C01817=1154.815,15.014,-48.250,179.930,6.144,149.128
C01818=1154.820,14.765,-48.236,179.927,6.143,149.129
C01819=1154.826,14.515,-48.222,179.924,6.142,149.129
C01820=1154.831,14.265,-48.208,179.922,6.141,149.130
C01821=1154.836,14.016,-48.194,179.919,6.140,149.130
C01822=1154.841,13.767,-48.180,179.917,6.140,149.131
C01823=1154.846,13.517,-48.166,179.915,6.139,149.131
C01824=1154.850,13.267,-48.152,179.911,6.138,149.132
C01825=1154.856,13.018,-48.139,179.909,6.137,149.133
C01826=1154.861,12.768,-48.125,179.906,6.137,149.133
C01827=1154.866,12.518,-48.110,179.904,6.136,149.134
C01828=1154.872,12.269,-48.096,179.902,6.135,149.134
C01829=1154.877,12.019,-48.083,179.899,6.134,149.135
C01830=1154.881,11.770,-48.069,179.896,6.133,149.136
C01831=1154.887,11.521,-48.055,179.894,6.132,149.136
C01832=1154.892,11.271,-48.041,179.891,6.132,149.137
C01833=1154.897,11.021,-48.027,179.889,6.131,149.137
C01834=1154.903,10.772,-48.013,179.887,6.131,149.138
C01835=1154.907,10.522,-48.000,179.884,6.129,149.138
C01836=1154.913,10.273,-47.987,179.881,6.129,149.139
C01837=1154.918,10.023,-47.972,179.879,6.128,149.139
C01838=1154.923,9.773,-47.958,179.876,6.127,149.140
C01839=1154.928,9.524,-47.945,179.874,6.127,149.141
C01840=1154.933,9.274,-47.931,179.871,6.125,149.141
C01841=1154.938,9.024,-47.917,179.869,6.125,149.142
C01842=1154.943,8.775,-47.904,179.866,6.124,149.142
C01843=1154.948,8.525,-47.890,179.864,6.123,149.143
C01844=1154.953,8.276,-47.876,179.861,6.123,149.144
C01845=1154.959,8.026,-47.862,179.859,6.122,149.144
C01846=1154.963,7.777,-47.849,179.856,6.121,149.145
C01847=1154.969,7.527,-47.836,179.854,6.120,149.145
C01848=1154.974,7.277,-47.821,179.851,6.119,149.146
C01849=1154.979,7.028,-47.807,179.849,6.119,149.146
C01850=1154.984,6.778,-47.794,179.846,6.118,149.147
C01851=1154.989,6.529,-47.781,179.844,6.117,149.147
C01852=1154.994,6.279,-47.767,179.841,6.116,149.148
C01853=1154.999,6.030,-47.754,179.839,6.115,149.149
C01854=1155.005,5.780,-47.740,179.836,6.115,149.149
C01855=1155.009,5.530,-47.726,179.834,6.114,149.150
C01856=1155.015,5.281,-47.713,179.831,6.114,149.150
C01857=1155.020,5.031,-47.699,179.829,6.113,149.151
C01858=1155.025,4.782,-47.686,179.826,6.111,149.152
C01859=1155.030,4.532,-47.672,179.824,6.111,149.152
C01860=1155.036,4.283,-47.659,179.821,6.110,149.153
C01861=1155.040,4.033,-47.645,179.819,6.109,149.153
C01862=1155.046,3.784,-47.632,179.816,6.109,149.154
C01863=1155.050,3.534,-47.618,179.814,6.108,149.154
C01864=1155.056,3.284,-47.605,179.811,6.108,149.155
C01865=1155.061,3.035,-47.591,179.808,6.106,149.155
C01866=1155.066,2.785,-47.578,179.806,6.106,149.156
C01867=1155.071,2.536,-47.564,179.804,6.105,149.157
C01868=1155.076,2.286,-47.551,179.801,6.104,149.157
C01869=1155.081,2.017,-47.536,179.799,6.104,149.158
C01870=1155.087,1.747,-47.522,179.796,6.102,149.158
C01871=1155.092,1.478,-47.507,179.793,6.102,149.159
C01872=1155.098,1.209,-47.494,179.790,6.101,149.160
C01873=1155.103,0.959,-47.479,179.788,6.101,149.160
C01874=1155.108,0.710,-47.467,179.785,6.100,149.161
C01875=1155.113,0.459,-47.453,179.783,6.099,149.161
C01876=1155.119,0.210,-47.439,179.780,6.098,149.162
C01877=1155.123,-0.040,-47.426,179.778,6.097,149.163
C01878=1155.129,-0.289,-47.413,179.775,6.097,149.163
C01879=1155.134,-0.539,-47.400,179.773,6.096,149.164
C01880=1155.139,-0.789,-47.386,179.770,6.096,149.164
C01881=1155.145,-1.038,-47.374,179.768,6.095,149.165
C01882=1155.149,-1.288,-47.360,179.766,6.094,149.166
C01883=1155.155,-1.537,-47.347,179.763,6.093,149.166
C01884=1155.160,-1.787,-47.333,179.760,6.092,149.167
C01885=1155.165,-2.036,-47.320,179.758,6.091,149.167
C01886=1155.169,-2.286,-47.307,179.755,6.091,149.168
C01887=1155.175,-2.536,-47.294,179.753,6.090,149.168
C01888=1155.180,-2.785,-47.281,179.750,6.090,149.169
C01889=1155.185,-3.035,-47.267,179.748,6.089,149.170
C01890=1155.190,-3.284,-47.254,179.746,6.088,149.170
C01891=1155.196,-3.534,-47.241,179.743,6.088,149.171
C01892=1155.201,-3.784,-47.228,179.741,6.087,149.171
C01893=1155.206,-4.033,-47.215,179.738,6.086,149.172
C01894=1155.211,-4.283,-47.201,179.735,6.085,149.173
C01895=1155.216,-4.532,-47.189,179.733,6.084,149.173
C01896=1155.221,-4.782,-47.175,179.731,6.084,149.174
C01897=1155.226,-5.032,-47.163,179.728,6.083,149.174
C01898=1155.232,-5.281,-47.149,179.726,6.083,149.175
C01899=1155.237,-5.531,-47.136,179.724,6.082,149.175
C01900=1155.241,-5.780,-47.123,179.721,6.081,149.176
C01901=1155.247,-6.029,-47.110,179.719,6.081,149.176
C01902=1155.252,-6.280,-47.097,179.716,6.080,149.177
C01903=1155.257,-6.529,-47.084,179.714,6.079,149.178
C01904=1155.263,-6.778,-47.071,179.711,6.079,149.178
C01905=1155.267,-7.028,-47.058,179.708,6.077,149.179
C01906=1155.273,-7.278,-47.045,179.706,6.077,149.179
C01907=1155.278,-7.527,-47.032,179.704,6.076,149.180
C01908=1155.283,-7.777,-47.019,179.701,6.076,149.181
C01909=1155.289,-8.027,-47.006,179.699,6.075,149.181
C01910=1155.294,-8.276,-46.993,179.696,6.074,149.182
C01911=1155.298,-8.526,-46.980,179.694,6.074,149.182
C01912=1155.303,-8.775,-46.967,179.691,6.073,149.183
C01913=1155.309,-9.025,-46.954,179.689,6.072,149.183
C01914=1155.314,-9.275,-46.941,179.686,6.072,149.184
C01915=1155.319,-9.524,-46.929,179.684,6.071,149.185
C01916=1155.325,-9.774,-46.915,179.682,6.071,149.185
C01917=1155.329,-10.024,-46.902,179.679,6.070,149.186
C01918=1155.334,-10.273,-46.890,179.677,6.069,149.186
C01919=1155.339,-10.522,-46.877,179.674,6.068,149.187
C01920=1155.345,-10.773,-46.864,179.671,6.067,149.188
C01921=1155.350,-11.022,-46.851,179.669,6.066,149.188
C01922=1155.355,-11.271,-46.838,179.666,6.066,149.189
C01923=1155.360,-11.521,-46.826,179.664,6.065,149.189
C01924=1155.365,-11.771,-46.812,179.662,6.065,149.190
C01925=1155.371,-12.021,-46.800,179.659,6.064,149.190
C01926=1155.376,-12.270,-46.788,179.657,6.064,149.191
C01927=1155.380,-12.520,-46.775,179.655,6.063,149.192
C01928=1155.386,-12.770,-46.762,179.652,6.062,149.192
C01929=1155.391,-13.019,-46.749,179.650,6.061,149.193
C01930=1155.396,-13.268,-46.736,179.647,6.061,149.193
C01931=1155.401,-13.519,-46.723,179.645,6.060,149.194
C01932=1155.406,-13.768,-46.711,179.642,6.060,149.195
C01933=1155.412,-14.017,-46.698,179.640,6.059,149.195
C01934=1155.417,-14.267,-46.685,179.637,6.059,149.196
C01935=1155.422,-14.517,-46.673,179.635,6.058,149.196
C01936=1155.427,-14.767,-46.660,179.633,6.057,149.197
C01937=1155.432,-15.016,-46.648,179.630,6.057,149.197
C01938=1155.437,-15.265,-46.635,179.628,6.056,149.198
C01939=1155.443,-15.515,-46.622,179.626,6.055,149.198
C01940=1155.448,-15.765,-46.609,179.623,6.055,149.199
C01941=1155.453,-16.015,-46.597,179.621,6.054,149.200
C01942=1155.458,-16.264,-46.584,179.618,6.054,149.200
C01943=1155.463,-16.514,-46.572,179.615,6.052,149.201
C01944=1155.468,-16.763,-46.559,179.613,6.052,149.201
C01945=1155.473,-17.014,-46.547,179.611,6.051,149.202
C01946=1155.478,-17.263,-46.534,179.608,6.050,149.203
C01947=1155.484,-17.512,-46.521,179.606,6.050,149.203
C01948=1155.489,-17.762,-46.509,179.603,6.049,149.204
C01949=1155.495,-18.012,-46.497,179.601,6.048,149.204
C01950=1155.500,-18.261,-46.484,179.598,6.048,149.205
C01951=1155.504,-18.511,-46.471,179.596,6.047,149.205
C01952=1155.510,-18.760,-46.458,179.593,6.047,149.206
C01953=1155.515,-19.010,-46.447,179.591,6.046,149.207
C01954=1155.520,-19.260,-46.434,179.588,6.045,149.207
C01955=1155.525,-19.509,-46.421,179.586,6.045,149.208
C01956=1155.531,-19.759,-46.409,179.584,6.044,149.208
C01957=1155.535,-20.009,-46.397,179.581,6.043,149.209
C01958=1155.540,-20.258,-46.384,179.579,6.043,149.210
C01959=1155.546,-20.508,-46.372,179.577,6.042,149.210
C01960=1155.551,-20.757,-46.359,179.574,6.042,149.211
C01961=1155.556,-21.007,-46.347,179.572,6.041,149.211
C01962=1155.562,-21.257,-46.334,179.569,6.040,149.212
C01963=1155.567,-21.506,-46.322,179.566,6.040,149.213
C01964=1155.572,-21.756,-46.309,179.564,6.039,149.213
C01965=1155.577,-22.006,-46.297,179.562,6.039,149.214
C01966=1155.582,-22.256,-46.284,179.559,6.038,149.214
C01967=1155.588,-22.506,-46.272,179.557,6.038,149.215
C01968=1155.593,-22.755,-46.260,179.555,6.037,149.215
C01969=1155.598,-23.004,-46.247,179.552,6.036,149.216
C01970=1155.603,-23.254,-46.235,179.550,6.036,149.217
C01971=1155.609,-23.503,-46.223,179.547,6.035,149.217
C01972=1155.613,-23.753,-46.211,179.545,6.034,149.218
C01973=1155.619,-24.023,-46.197,179.542,6.034,149.219
C01974=1155.625,-24.293,-46.185,179.540,6.033,149.219
C01975=1155.630,-24.563,-46.172,179.537,6.033,149.220
C01976=1155.636,-24.833,-46.157,179.535,6.032,149.220
C01977=1155.641,-25.083,-46.146,179.533,6.031,149.221
C01978=1155.646,-25.332,-46.133,179.530,6.031,149.222
C01979=1155.651,-25.582,-46.122,179.528,6.030,149.222
C01980=1155.656,-25.831,-46.109,179.525,6.030,149.223
C01981=1155.662,-26.081,-46.097,179.523,6.029,149.223
C01982=1155.667,-26.331,-46.084,179.520,6.029,149.224
C01983=1155.672,-26.581,-46.073,179.518,6.028,149.224
C01984=1155.677,-26.830,-46.060,179.515,6.027,149.225
C01985=1155.683,-27.080,-46.048,179.513,6.027,149.226
C01986=1155.688,-27.330,-46.036,179.511,6.026,149.226
C01987=1155.693,-27.579,-46.024,179.508,6.025,149.227
C01988=1155.698,-27.829,-46.012,179.506,6.025,149.227
C01989=1155.703,-28.078,-46.000,179.504,6.024,149.228
C01990=1155.709,-28.328,-45.988,179.501,6.024,149.229
C01991=1155.714,-28.577,-45.975,179.499,6.023,149.229
C01992=1155.719,-28.827,-45.963,179.496,6.022,149.230
C01993=1155.725,-29.077,-45.951,179.494,6.022,149.230
C01994=1155.729,-29.326,-45.939,179.492,6.022,149.231
C01995=1155.734,-29.576,-45.928,179.490,6.021,149.231
C01996=1155.740,-29.826,-45.916,179.487,6.021,149.232
C01997=1155.745,-30.075,-45.903,179.485,6.020,149.233
C01998=1155.750,-30.325,-45.891,179.482,6.020,149.233
C01999=1155.755,-30.575,-45.880,179.480,6.019,149.234
C02000=1155.760,-30.824,-45.867,179.477,6.018,149.234
C02001=1155.766,-31.074,-45.855,179.475,6.018,149.235
C02002=1155.771,-31.324,-45.844,179.472,6.017,149.236
C02003=1155.776,-31.573,-45.831,179.470,6.016,149.236
C02004=1155.781,-31.823,-45.820,179.468,6.016,149.237
C02005=1155.786,-32.073,-45.808,179.465,6.015,149.237
C02006=1155.791,-32.322,-45.795,179.463,6.015,149.238
C02007=1155.797,-32.572,-45.783,179.461,6.014,149.238
C02008=1155.802,-32.822,-45.772,179.458,6.013,149.239
C02009=1155.807,-33.072,-45.760,179.456,6.013,149.240
C02010=1155.812,-33.321,-45.747,179.453,6.012,149.240
C02011=1155.818,-33.571,-45.736,179.451,6.012,149.241
C02012=1155.822,-33.821,-45.724,179.449,6.012,149.241
C02013=1155.828,-34.071,-45.712,179.447,6.011,149.242
C02014=1155.833,-34.320,-45.700,179.444,6.011,149.243
C02015=1155.838,-34.570,-45.688,179.442,6.010,149.243
C02016=1155.843,-34.820,-45.677,179.439,6.009,149.244
C02017=1155.849,-35.069,-45.665,179.437,6.009,149.244
C02018=1155.854,-35.319,-45.653,179.434,6.008,149.245
C02019=1155.859,-35.568,-45.641,179.432,6.007,149.245
C02020=1155.864,-35.818,-45.629,179.429,6.007,149.246
C02021=1155.870,-36.068,-45.617,179.427,6.006,149.247
C02022=1155.875,-36.317,-45.606,179.425,6.006,149.247
C02023=1155.880,-36.567,-45.594,179.423,6.006,149.248
C02024=1155.885,-36.817,-45.582,179.420,6.005,149.248
C02025=1155.891,-37.067,-45.571,179.418,6.005,149.249
C02026=1155.896,-37.315,-45.559,179.416,6.004,149.249
C02027=1155.901,-37.565,-45.547,179.413,6.003,149.250
C02028=1155.906,-37.815,-45.535,179.411,6.003,149.251
C02029=1155.911,-38.065,-45.524,179.408,6.002,149.251
C02030=1155.917,-38.315,-45.512,179.406,6.001,149.252
C02031=1155.921,-38.564,-45.501,179.404,6.001,149.252
C02032=1155.927,-38.814,-45.489,179.401,6.000,149.253
C02033=1155.932,-39.064,-45.477,179.399,6.000,149.254
C02034=1155.937,-39.313,-45.466,179.397,6.000,149.254
C02035=1155.943,-39.563,-45.454,179.394,5.999,149.255
C02036=1155.948,-39.813,-45.442,179.392,5.998,149.255
C02037=1155.953,-40.063,-45.431,179.390,5.998,149.256
C02038=1155.958,-40.313,-45.419,179.387,5.997,149.256
C02039=1155.963,-40.562,-45.408,179.385,5.997,149.257
C02040=1155.969,-40.811,-45.396,179.383,5.996,149.258
C02041=1155.975,-41.061,-45.384,179.380,5.996,149.258
C02042=1155.979,-41.310,-45.372,179.378,5.995,149.259
C02043=1155.985,-41.561,-45.361,179.376,5.995,149.260
C02044=1155.989,-41.811,-45.350,179.373,5.994,149.260
C02045=1155.995,-42.060,-45.338,179.371,5.994,149.261
C02046=1156.000,-42.309,-45.327,179.369,5.993,149.261
C02047=1156.006,-42.559,-45.315,179.366,5.993,149.262
C02048=1156.010,-42.809,-45.304,179.364,5.992,149.262
C02049=1156.016,-43.059,-45.292,179.361,5.992,149.263
C02050=1156.021,-43.308,-45.281,179.359,5.991,149.264
C02051=1156.026,-43.558,-45.269,179.357,5.991,149.264
C02052=1156.031,-43.807,-45.258,179.355,5.990,149.265
C02053=1156.036,-44.057,-45.246,179.352,5.990,149.265
C02054=1156.041,-44.307,-45.235,179.350,5.989,149.266
C02055=1156.047,-44.556,-45.223,179.348,5.988,149.266
C02056=1156.052,-44.806,-45.212,179.345,5.988,149.267
C02057=1156.057,-45.056,-45.200,179.343,5.987,149.268
C02058=1156.062,-45.306,-45.189,179.340,5.987,149.268
C02059=1156.068,-45.555,-45.178,179.339,5.987,149.269
C02060=1156.073,-45.805,-45.167,179.336,5.986,149.269
C02061=1156.078,-46.055,-45.155,179.334,5.986,149.270
C02062=1156.083,-46.304,-45.143,179.331,5.985,149.271
C02063=1156.089,-46.554,-45.132,179.329,5.984,149.271
C02064=1156.094,-46.803,-45.121,179.326,5.984,149.272
C02065=1156.100,-47.054,-45.109,179.324,5.983,149.272
C02066=1156.104,-47.303,-45.098,179.322,5.984,149.273
C02067=1156.110,-47.553,-45.087,179.320,5.983,149.273
C02068=1156.115,-47.802,-45.075,179.317,5.982,149.274
C02069=1156.120,-48.052,-45.064,179.315,5.982,149.275
C02070=1156.125,-48.303,-45.053,179.313,5.981,149.275
C02071=1156.131,-48.551,-45.042,179.310,5.980,149.276
C02072=1156.136,-48.801,-45.030,179.308,5.980,149.276
C02073=1156.141,-49.051,-45.019,179.306,5.980,149.277
C02074=1156.146,-49.300,-45.008,179.304,5.979,149.277
C02075=1156.152,-49.550,-44.997,179.301,5.979,149.278
C02076=1156.157,-49.800,-44.985,179.299,5.978,149.279
C02077=1156.163,-50.070,-44.974,179.296,5.978,149.279
C02078=1156.168,-50.341,-44.961,179.293,5.977,149.280
C02079=1156.174,-50.612,-44.949,179.291,5.976,149.281
C02080=1156.180,-50.882,-44.936,179.288,5.976,149.281
C02081=1156.185,-51.132,-44.926,179.286,5.975,149.282
C02082=1156.190,-51.382,-44.915,179.284,5.976,149.282
C02083=1156.196,-51.631,-44.903,179.282,5.975,149.283
C02084=1156.201,-51.881,-44.892,179.279,5.974,149.284
C02085=1156.205,-52.131,-44.881,179.277,5.974,149.284
C02086=1156.211,-52.380,-44.870,179.275,5.973,149.285
C02087=1156.216,-52.630,-44.859,179.272,5.972,149.285
C02088=1156.221,-52.880,-44.848,179.270,5.973,149.286
C02089=1156.227,-53.129,-44.836,179.268,5.972,149.286
C02090=1156.232,-53.380,-44.826,179.265,5.972,149.287
C02091=1156.237,-53.629,-44.814,179.263,5.971,149.288
C02092=1156.243,-53.878,-44.803,179.261,5.970,149.288
C02093=1156.248,-54.129,-44.792,179.258,5.970,149.289
C02094=1156.253,-54.378,-44.781,179.257,5.970,149.289
C02095=1156.258,-54.628,-44.771,179.254,5.969,149.290
C02096=1156.264,-54.878,-44.759,179.252,5.969,149.290
C02097=1156.269,-55.127,-44.748,179.249,5.968,149.291
C02098=1156.274,-55.377,-44.737,179.247,5.967,149.292
C02099=1156.279,-55.627,-44.726,179.245,5.968,149.292
C02100=1156.285,-55.876,-44.715,179.243,5.967,149.293
C02101=1156.290,-56.126,-44.704,179.240,5.967,149.294
C02102=1156.295,-56.376,-44.694,179.238,5.966,149.294
C02103=1156.300,-56.625,-44.683,179.236,5.965,149.294
C02104=1156.305,-56.875,-44.671,179.234,5.965,149.295
C02105=1156.311,-57.125,-44.660,179.232,5.965,149.296
C02106=1156.316,-57.374,-44.649,179.229,5.964,149.296
C02107=1156.321,-57.624,-44.639,179.227,5.963,149.297
C02108=1156.326,-57.873,-44.628,179.224,5.963,149.298
C02109=1156.332,-58.124,-44.617,179.222,5.962,149.298
C02110=1156.337,-58.373,-44.606,179.220,5.963,149.299
C02111=1156.342,-58.623,-44.595,179.218,5.962,149.299
C02112=1156.347,-58.872,-44.584,179.215,5.961,149.300
C02113=1156.352,-59.122,-44.574,179.213,5.961,149.300
C02114=1156.358,-59.373,-44.562,179.211,5.961,149.301
C02115=1156.363,-59.622,-44.551,179.208,5.960,149.302
C02116=1156.368,-59.872,-44.541,179.206,5.959,149.302
C02117=1156.374,-60.121,-44.530,179.204,5.959,149.303
C02118=1156.379,-60.371,-44.519,179.201,5.958,149.303
C02119=1156.384,-60.620,-44.508,179.199,5.959,149.304
C02120=1156.389,-60.870,-44.498,179.197,5.958,149.304
C02121=1156.395,-61.120,-44.487,179.195,5.957,149.305
C02122=1156.400,-61.370,-44.476,179.192,5.957,149.306
C02123=1156.405,-61.619,-44.466,179.190,5.956,149.306
C02124=1156.410,-61.869,-44.454,179.188,5.956,149.307
C02125=1156.416,-62.119,-44.444,179.186,5.956,149.307
C02126=1156.421,-62.369,-44.433,179.183,5.955,149.308
C02127=1156.425,-62.619,-44.422,179.181,5.954,149.308
C02128=1156.431,-62.868,-44.412,179.179,5.954,149.309
C02129=1156.437,-63.119,-44.401,179.177,5.954,149.310
C02130=1156.442,-63.368,-44.390,179.174,5.953,149.310
C02131=1156.447,-63.618,-44.379,179.172,5.953,149.311
C02132=1156.453,-63.867,-44.369,179.170,5.952,149.311
C02133=1156.457,-64.117,-44.358,179.168,5.952,149.312
C02134=1156.463,-64.367,-44.348,179.165,5.952,149.312
C02135=1156.468,-64.617,-44.337,179.163,5.951,149.313
C02136=1156.473,-64.866,-44.326,179.161,5.950,149.314
C02137=1156.478,-65.116,-44.316,179.159,5.950,149.314
C02138=1156.484,-65.365,-44.305,179.156,5.950,149.315
C02139=1156.489,-65.614,-44.294,179.154,5.949,149.315
C02140=1156.494,-65.865,-44.284,179.151,5.949,149.316
C02141=1156.500,-66.114,-44.274,179.150,5.949,149.317
C02142=1156.505,-66.364,-44.263,179.148,5.948,149.317
C02143=1156.510,-66.613,-44.252,179.145,5.948,149.318
C02144=1156.515,-66.864,-44.242,179.143,5.947,149.318
C02145=1156.521,-67.113,-44.231,179.141,5.947,149.319
C02146=1156.526,-67.363,-44.221,179.138,5.947,149.319
C02147=1156.532,-67.613,-44.209,179.136,5.946,149.320
C02148=1156.537,-67.863,-44.199,179.134,5.945,149.321
C02149=1156.542,-68.112,-44.188,179.132,5.945,149.321
C02150=1156.548,-68.362,-44.178,179.129,5.945,149.322
C02151=1156.552,-68.612,-44.168,179.127,5.944,149.322
C02152=1156.558,-68.861,-44.158,179.124,5.944,149.323
C02153=1156.562,-69.111,-44.147,179.123,5.944,149.323
C02154=1156.568,-69.361,-44.137,179.120,5.943,149.324
C02155=1156.574,-69.610,-44.126,179.118,5.943,149.325
C02156=1156.579,-69.860,-44.116,179.116,5.942,149.325
C02157=1156.584,-70.110,-44.106,179.114,5.942,149.326
C02158=1156.589,-70.360,-44.095,179.112,5.942,149.326
C02159=1156.594,-70.609,-44.084,179.109,5.941,149.327
C02160=1156.599,-70.859,-44.074,179.107,5.940,149.327
C02161=1156.605,-71.109,-44.063,179.105,5.940,149.328
C02162=1156.611,-71.358,-44.053,179.102,5.940,149.329
C02163=1156.616,-71.609,-44.043,179.100,5.939,149.329
C02164=1156.621,-71.858,-44.032,179.098,5.939,149.330
C02165=1156.627,-72.108,-44.022,179.096,5.939,149.330
C02166=1156.632,-72.358,-44.012,179.094,5.938,149.331
C02167=1156.637,-72.608,-44.001,179.091,5.938,149.332
C02168=1156.642,-72.858,-43.991,179.090,5.938,149.332
C02169=1156.648,-73.107,-43.981,179.087,5.937,149.333
C02170=1156.653,-73.356,-43.970,179.085,5.937,149.333
C02171=1156.658,-73.606,-43.960,179.083,5.936,149.334
C02172=1156.663,-73.856,-43.949,179.080,5.936,149.334
C02173=1156.669,-74.105,-43.939,179.078,5.935,149.335
C02174=1156.674,-74.356,-43.929,179.076,5.935,149.336
C02175=1156.679,-74.605,-43.918,179.074,5.935,149.336
C02176=1156.685,-74.855,-43.908,179.071,5.935,149.337
C02177=1156.690,-75.105,-43.898,179.069,5.934,149.337
C02178=1156.695,-75.354,-43.888,179.067,5.933,149.338
C02179=1156.700,-75.604,-43.878,179.065,5.933,149.338
C02180=1156.705,-75.854,-43.867,179.063,5.933,149.339
C02181=1156.712,-76.125,-43.856,179.060,5.932,149.340
C02182=1156.717,-76.396,-43.845,179.058,5.932,149.340
C02183=1156.723,-76.668,-43.834,179.055,5.931,149.341
C02184=1156.729,-76.939,-43.824,179.054,5.931,149.341
C02185=1156.734,-77.189,-43.813,179.051,5.931,149.342
C02186=1156.740,-77.439,-43.803,179.049,5.930,149.342
C02187=1156.745,-77.688,-43.793,179.046,5.930,149.343
C02188=1156.750,-77.938,-43.783,179.044,5.930,149.344
C02189=1156.755,-78.188,-43.773,179.042,5.929,149.344
C02190=1156.761,-78.437,-43.762,179.040,5.928,149.345
C02191=1156.766,-78.687,-43.752,179.038,5.928,149.345
C02192=1156.771,-78.937,-43.742,179.035,5.928,149.346
C02193=1156.776,-79.186,-43.732,179.033,5.927,149.347
C02194=1156.782,-79.436,-43.722,179.031,5.927,149.347
C02195=1156.787,-79.687,-43.712,179.029,5.927,149.348
C02196=1156.793,-79.936,-43.702,179.027,5.926,149.348
C02197=1156.798,-80.185,-43.692,179.024,5.926,149.349
C02198=1156.803,-80.435,-43.682,179.022,5.926,149.349
C02199=1156.808,-80.685,-43.671,179.020,5.925,149.350
C02200=1156.814,-80.935,-43.661,179.017,5.925,149.351
C02201=1156.819,-81.184,-43.651,179.016,5.925,149.351
C02202=1156.825,-81.434,-43.642,179.014,5.924,149.352
C02203=1156.830,-81.684,-43.631,179.011,5.924,149.352
C02204=1156.835,-81.934,-43.621,179.009,5.924,149.353
C02205=1156.840,-82.183,-43.612,179.007,5.923,149.353
C02206=1156.846,-82.433,-43.601,179.005,5.922,149.354
C02207=1156.851,-82.684,-43.592,179.003,5.922,149.354
C02208=1156.856,-82.933,-43.582,179.000,5.922,149.355
C02209=1156.861,-83.182,-43.572,178.998,5.921,149.356
C02210=1156.867,-83.432,-43.561,178.997,5.921,149.356
C02211=1156.872,-83.682,-43.553,178.994,5.921,149.357
C02212=1156.877,-83.932,-43.542,178.992,5.920,149.357
C02213=1156.883,-84.182,-43.532,178.990,5.921,149.358
C02214=1156.888,-84.431,-43.522,178.987,5.920,149.358
C02215=1156.894,-84.681,-43.513,178.985,5.919,149.359
C02216=1156.899,-84.931,-43.502,178.983,5.919,149.360
C02217=1156.903,-85.180,-43.492,178.981,5.919,149.360
C02218=1156.909,-85.430,-43.482,178.979,5.918,149.361
C02219=1156.915,-85.680,-43.473,178.977,5.918,149.361
C02220=1156.920,-85.929,-43.463,178.974,5.918,149.362
C02221=1156.925,-86.180,-43.453,178.972,5.917,149.362
C02222=1156.931,-86.430,-43.443,178.970,5.917,149.363
C02223=1156.935,-86.679,-43.434,178.968,5.916,149.364
C02224=1156.941,-86.929,-43.423,178.966,5.916,149.364
C02225=1156.946,-87.178,-43.414,178.964,5.916,149.365
C02226=1156.952,-87.428,-43.404,178.962,5.915,149.365
C02227=1156.957,-87.678,-43.394,178.959,5.915,149.366
C02228=1156.962,-87.928,-43.385,178.957,5.915,149.366
C02229=1156.968,-88.178,-43.375,178.955,5.914,149.367
C02230=1156.972,-88.427,-43.365,178.952,5.914,149.368
C02231=1156.978,-88.677,-43.355,178.951,5.914,149.368
C02232=1156.983,-88.926,-43.346,178.949,5.913,149.369
C02233=1156.988,-89.176,-43.335,178.946,5.913,149.369
C02234=1156.994,-89.427,-43.326,178.944,5.913,149.370
C02235=1156.999,-89.676,-43.316,178.942,5.912,149.370
C02236=1157.005,-89.926,-43.307,178.939,5.911,149.371
C02237=1157.010,-90.175,-43.297,178.938,5.912,149.371
C02238=1157.015,-90.425,-43.287,178.936,5.911,149.372
C02239=1157.021,-90.675,-43.278,178.933,5.910,149.373
C02240=1157.026,-90.925,-43.267,178.931,5.910,149.373
C02241=1157.031,-91.175,-43.258,178.929,5.910,149.374
C02242=1157.036,-91.424,-43.248,178.927,5.910,149.374
C02243=1157.041,-91.674,-43.239,178.925,5.909,149.375
C02244=1157.047,-91.924,-43.229,178.923,5.908,149.375
C02245=1157.052,-92.174,-43.220,178.921,5.909,149.376
C02246=1157.058,-92.423,-43.210,178.919,5.908,149.376
C02247=1157.064,-92.673,-43.201,178.916,5.907,149.377
C02248=1157.069,-92.922,-43.191,178.914,5.908,149.378
C02249=1157.074,-93.173,-43.180,178.912,5.907,149.378
C02250=1157.079,-93.423,-43.171,178.910,5.906,149.379
C02251=1157.084,-93.672,-43.162,178.908,5.907,149.379
C02252=1157.090,-93.922,-43.152,178.906,5.906,149.380
C02253=1157.095,-94.172,-43.143,178.904,5.906,149.380
C02254=1157.100,-94.421,-43.133,178.901,5.906,149.381
C02255=1157.105,-94.671,-43.124,178.899,5.905,149.381
C02256=1157.111,-94.921,-43.114,178.898,5.905,149.382
C02257=1157.116,-95.171,-43.105,178.895,5.904,149.383
C02258=1157.122,-95.420,-43.095,178.893,5.904,149.383
C02259=1157.127,-95.670,-43.086,178.891,5.904,149.384
C02260=1157.133,-95.920,-43.076,178.888,5.903,149.384
C02261=1157.138,-96.169,-43.067,178.887,5.903,149.385
C02262=1157.144,-96.420,-43.057,178.885,5.903,149.385
C02263=1157.148,-96.669,-43.048,178.882,5.902,149.386
C02264=1157.153,-96.919,-43.039,178.880,5.902,149.387
C02265=1157.159,-97.169,-43.028,178.878,5.901,149.387
C02266=1157.164,-97.419,-43.020,178.876,5.902,149.388
C02267=1157.170,-97.669,-43.010,178.874,5.901,149.388
C02268=1157.175,-97.918,-43.000,178.872,5.900,149.389
C02269=1157.180,-98.168,-42.992,178.870,5.901,149.389
C02270=1157.185,-98.418,-42.981,178.867,5.900,149.390
C02271=1157.191,-98.667,-42.972,178.865,5.899,149.390
C02272=1157.196,-98.918,-42.963,178.864,5.899,149.391
C02273=1157.201,-99.167,-42.953,178.861,5.899,149.392
C02274=1157.206,-99.417,-42.944,178.859,5.899,149.392
C02275=1157.212,-99.667,-42.935,178.857,5.898,149.393
C02276=1157.217,-99.916,-42.925,178.854,5.898,149.393
C02277=1157.223,-100.166,-42.916,178.853,5.898,149.394
C02278=1157.228,-100.416,-42.907,178.851,5.897,149.394
C02279=1157.233,-100.665,-42.897,178.849,5.897,149.395
C02280=1157.239,-100.915,-42.888,178.846,5.897,149.395
C02281=1157.244,-101.165,-42.879,178.844,5.896,149.396
C02282=1157.249,-101.415,-42.870,178.842,5.896,149.397
C02283=1157.255,-101.665,-42.860,178.840,5.896,149.397
C02284=1157.260,-101.915,-42.851,178.838,5.896,149.398
C02285=1157.266,-102.186,-42.841,178.836,5.895,149.398
C02286=1157.272,-102.458,-42.832,178.833,5.894,149.399
C02287=1157.278,-102.730,-42.821,178.831,5.894,149.400
C02288=1157.284,-103.002,-42.810,178.829,5.894,149.400
C02289=1157.289,-103.252,-42.802,178.827,5.893,149.400
C02290=1157.294,-103.502,-42.793,178.825,5.894,149.401
C02291=1157.299,-103.751,-42.783,178.823,5.893,149.402
C02292=1157.305,-104.002,-42.774,178.821,5.892,149.402
C02293=1157.310,-104.251,-42.765,178.818,5.893,149.403
C02294=1157.315,-104.501,-42.756,178.816,5.892,149.403
C02295=1157.320,-104.750,-42.746,178.815,5.892,149.404
C02296=1157.326,-105.001,-42.737,178.812,5.891,149.404
C02297=1157.331,-105.250,-42.728,178.810,5.891,149.405
C02298=1157.336,-105.500,-42.719,178.808,5.891,149.406
C02299=1157.342,-105.749,-42.710,178.806,5.890,149.406
C02300=1157.348,-106.000,-42.701,178.804,5.890,149.406
C02301=1157.353,-106.249,-42.691,178.802,5.890,149.407
C02302=1157.358,-106.499,-42.682,178.800,5.890,149.408
C02303=1157.363,-106.749,-42.673,178.798,5.889,149.408
C02304=1157.369,-106.999,-42.664,178.795,5.889,149.409
C02305=1157.374,-107.249,-42.655,178.794,5.889,149.409
C02306=1157.379,-107.498,-42.646,178.791,5.888,149.410
C02307=1157.385,-107.748,-42.637,178.790,5.888,149.410
C02308=1157.390,-107.998,-42.627,178.787,5.888,149.411
C02309=1157.395,-108.248,-42.618,178.786,5.888,149.412
C02310=1157.401,-108.498,-42.609,178.783,5.887,149.412
C02311=1157.406,-108.747,-42.601,178.781,5.886,149.413
C02312=1157.411,-108.997,-42.592,178.779,5.887,149.413
C02313=1157.417,-109.247,-42.582,178.777,5.886,149.414
C02314=1157.423,-109.497,-42.573,178.775,5.886,149.414
C02315=1157.428,-109.746,-42.565,178.773,5.885,149.415
C02316=1157.433,-109.996,-42.556,178.771,5.885,149.415
C02317=1157.438,-110.246,-42.547,178.769,5.885,149.416
C02318=1157.443,-110.496,-42.538,178.767,5.884,149.416
C02319=1157.450,-110.745,-42.529,178.765,5.884,149.417
C02320=1157.455,-110.995,-42.520,178.762,5.884,149.418
C02321=1157.460,-111.245,-42.511,178.761,5.884,149.418
C02322=1157.465,-111.495,-42.502,178.759,5.883,149.419
C02323=1157.470,-111.745,-42.493,178.757,5.883,149.419
C02324=1157.476,-111.995,-42.484,178.754,5.883,149.420
C02325=1157.481,-112.245,-42.475,178.753,5.883,149.420
C02326=1157.487,-112.494,-42.466,178.751,5.882,149.421
C02327=1157.492,-112.744,-42.457,178.748,5.881,149.421
C02328=1157.498,-112.994,-42.448,178.746,5.882,149.422
C02329=1157.503,-113.244,-42.439,178.744,5.881,149.422
C02330=1157.508,-113.493,-42.431,178.742,5.881,149.423
C02331=1157.513,-113.743,-42.422,178.740,5.880,149.423
C02332=1157.519,-113.992,-42.413,178.738,5.880,149.424
C02333=1157.524,-114.242,-42.404,178.736,5.880,149.425
C02334=1157.529,-114.492,-42.395,178.734,5.880,149.425
C02335=1157.535,-114.742,-42.386,178.732,5.879,149.426
C02336=1157.540,-114.992,-42.377,178.730,5.879,149.426
C02337=1157.546,-115.241,-42.368,178.728,5.879,149.427
C02338=1157.551,-115.491,-42.360,178.726,5.878,149.427
C02339=1157.556,-115.741,-42.351,178.724,5.878,149.428
C02340=1157.561,-115.991,-42.342,178.721,5.878,149.428
C02341=1157.567,-116.241,-42.333,178.720,5.878,149.429
C02342=1157.572,-116.490,-42.324,178.718,5.877,149.429
C02343=1157.578,-116.740,-42.316,178.716,5.877,149.430
C02344=1157.583,-116.990,-42.307,178.714,5.876,149.430
C02345=1157.588,-117.240,-42.298,178.712,5.877,149.431
C02346=1157.593,-117.490,-42.289,178.710,5.876,149.432
C02347=1157.599,-117.739,-42.281,178.708,5.876,149.432
C02348=1157.604,-117.989,-42.272,178.706,5.875,149.433
C02349=1157.609,-118.239,-42.263,178.704,5.875,149.433
C02350=1157.615,-118.489,-42.255,178.702,5.875,149.434
C02351=1157.621,-118.738,-42.246,178.700,5.875,149.434
C02352=1157.626,-118.988,-42.238,178.698,5.874,149.435
C02353=1157.631,-119.238,-42.229,178.696,5.874,149.435
C02354=1157.636,-119.488,-42.220,178.693,5.874,149.436
C02355=1157.642,-119.737,-42.211,178.691,5.873,149.436
C02356=1157.647,-119.987,-42.203,178.690,5.873,149.437
C02357=1157.653,-120.237,-42.194,178.687,5.872,149.437
C02358=1157.658,-120.487,-42.185,178.686,5.872,149.438
C02359=1157.664,-120.736,-42.177,178.683,5.872,149.439
C02360=1157.669,-120.986,-42.168,178.682,5.872,149.439
C02361=1157.674,-121.237,-42.160,178.679,5.871,149.440
C02362=1157.679,-121.487,-42.151,178.678,5.871,149.440
C02363=1157.685,-121.736,-42.142,178.676,5.870,149.441
C02364=1157.690,-121.985,-42.133,178.674,5.871,149.441
C02365=1157.696,-122.236,-42.125,178.671,5.870,149.442
C02366=1157.701,-122.486,-42.116,178.670,5.870,149.442
C02367=1157.707,-122.735,-42.108,178.668,5.869,149.443
C02368=1157.712,-122.985,-42.099,178.666,5.869,149.443
C02369=1157.717,-123.235,-42.091,178.663,5.869,149.444
C02370=1157.723,-123.484,-42.082,178.662,5.869,149.444
C02371=1157.728,-123.734,-42.074,178.659,5.868,149.445
C02372=1157.733,-123.984,-42.066,178.658,5.868,149.445
C02373=1157.738,-124.234,-42.057,178.656,5.868,149.446
C02374=1157.744,-124.483,-42.048,178.654,5.868,149.446
C02375=1157.749,-124.733,-42.039,178.651,5.867,149.447
C02376=1157.755,-124.984,-42.031,178.650,5.867,149.448
C02377=1157.760,-125.233,-42.023,178.648,5.867,149.448
C02378=1157.766,-125.483,-42.014,178.646,5.867,149.449
C02379=1157.771,-125.733,-42.005,178.644,5.866,149.449
C02380=1157.777,-125.982,-41.997,178.642,5.866,149.450
C02381=1157.781,-126.232,-41.989,178.640,5.866,149.450
C02382=1157.787,-126.482,-41.980,178.638,5.866,149.451
C02383=1157.792,-126.732,-41.972,178.636,5.865,149.451
C02384=1157.798,-126.982,-41.964,178.634,5.865,149.452
C02385=1157.803,-127.232,-41.955,178.632,5.864,149.452
C02386=1157.809,-127.481,-41.946,178.630,5.865,149.453
C02387=1157.814,-127.732,-41.938,178.628,5.864,149.453
C02388=1157.819,-127.981,-41.930,178.626,5.864,149.454
C02389=1157.399,-127.992,-41.972,178.622,5.867,149.456
C02390=1157.393,-127.742,-41.980,178.624,5.868,149.455
C02391=1157.388,-127.493,-41.989,178.626,5.867,149.455
C02392=1157.382,-127.242,-41.997,178.629,5.868,149.454
C02393=1157.376,-126.993,-42.005,178.630,5.868,149.454
C02394=1157.371,-126.743,-42.014,178.632,5.869,149.453
C02395=1157.366,-126.493,-42.022,178.634,5.869,149.453
C02396=1157.361,-126.244,-42.030,178.636,5.870,149.452
C02397=1157.356,-125.994,-42.039,178.638,5.869,149.451
C02398=1157.350,-125.743,-42.048,178.641,5.870,149.451
C02399=1157.344,-125.494,-42.056,178.642,5.870,149.450
C02400=1157.339,-125.244,-42.065,178.644,5.871,149.450
C02401=1157.334,-124.994,-42.073,178.646,5.871,149.449
C02402=1157.328,-124.745,-42.082,178.648,5.871,149.449
C02403=1157.323,-124.495,-42.091,178.650,5.871,149.448
C02404=1157.318,-124.245,-42.098,178.652,5.872,149.448
C02405=1157.312,-123.996,-42.107,178.654,5.872,149.447
C02406=1157.307,-123.746,-42.116,178.656,5.872,149.447
C02407=1157.302,-123.495,-42.124,178.658,5.872,149.446
C02408=1157.296,-123.246,-42.132,178.660,5.873,149.446
C02409=1157.291,-122.996,-42.141,178.662,5.873,149.445
C02410=1157.285,-122.746,-42.150,178.664,5.873,149.445
C02411=1157.280,-122.496,-42.158,178.666,5.873,149.444
C02412=1157.274,-122.247,-42.167,178.668,5.874,149.444
C02413=1157.269,-121.997,-42.176,178.670,5.874,149.443
C02414=1157.264,-121.747,-42.185,178.672,5.874,149.442
C02415=1157.258,-121.497,-42.192,178.674,5.874,149.442
C02416=1157.253,-121.248,-42.201,178.676,5.875,149.441
C02417=1157.247,-120.998,-42.210,178.678,5.875,149.441
C02418=1157.242,-120.748,-42.219,178.680,5.876,149.440
C02419=1157.237,-120.498,-42.226,178.682,5.875,149.440
C02420=1157.232,-120.249,-42.235,178.684,5.876,149.439
C02421=1157.227,-119.999,-42.244,178.686,5.876,149.439
C02422=1157.221,-119.749,-42.253,178.688,5.877,149.438
C02423=1157.216,-119.500,-42.262,178.690,5.877,149.438
C02424=1157.210,-119.249,-42.270,178.692,5.877,149.437
C02425=1157.205,-118.999,-42.279,178.694,5.877,149.437
C02426=1157.200,-118.749,-42.288,178.696,5.878,149.436
C02427=1157.194,-118.500,-42.296,178.698,5.878,149.436
C02428=1157.189,-118.251,-42.305,178.700,5.879,149.435
C02429=1157.184,-118.001,-42.314,178.703,5.879,149.434
C02430=1157.178,-117.750,-42.322,178.704,5.879,149.434
C02431=1157.173,-117.500,-42.331,178.706,5.880,149.433
C02432=1157.167,-117.251,-42.339,178.708,5.880,149.433
C02433=1157.161,-117.001,-42.349,178.711,5.880,149.432
C02434=1157.156,-116.751,-42.358,178.712,5.880,149.432
C02435=1157.151,-116.501,-42.367,178.714,5.881,149.431
C02436=1157.145,-116.252,-42.375,178.716,5.881,149.431
C02437=1157.140,-116.002,-42.384,178.718,5.882,149.430
C02438=1157.135,-115.752,-42.392,178.720,5.881,149.430
C02439=1157.130,-115.502,-42.401,178.722,5.882,149.429
C02440=1157.124,-115.252,-42.410,178.724,5.882,149.429
C02441=1157.119,-115.003,-42.419,178.726,5.883,149.428
C02442=1157.113,-114.753,-42.428,178.728,5.882,149.427
C02443=1157.108,-114.503,-42.437,178.731,5.883,149.427
C02444=1157.103,-114.253,-42.445,178.733,5.884,149.426
C02445=1157.098,-114.004,-42.454,178.734,5.884,149.426
C02446=1157.093,-113.754,-42.463,178.737,5.884,149.425
C02447=1157.086,-113.504,-42.472,178.739,5.884,149.425
C02448=1157.081,-113.254,-42.481,178.741,5.885,149.424
C02449=1157.076,-113.005,-42.490,178.742,5.885,149.424
C02450=1157.071,-112.755,-42.499,178.745,5.886,149.423
C02451=1157.066,-112.505,-42.508,178.747,5.885,149.423
C02452=1157.060,-112.255,-42.517,178.749,5.886,149.422
C02453=1157.055,-112.006,-42.525,178.751,5.887,149.422
C02454=1157.050,-111.756,-42.534,178.753,5.887,149.421
C02455=1157.044,-111.506,-42.544,178.755,5.887,149.420
C02456=1157.038,-111.256,-42.553,178.757,5.887,149.420
C02457=1157.033,-111.006,-42.562,178.759,5.888,149.419
C02458=1157.028,-110.756,-42.570,178.761,5.888,149.419
C02459=1157.022,-110.507,-42.579,178.763,5.888,149.418
C02460=1157.017,-110.257,-42.588,178.765,5.888,149.418
C02461=1157.011,-110.007,-42.597,178.767,5.889,149.417
C02462=1157.006,-109.757,-42.606,178.769,5.889,149.417
C02463=1157.001,-109.507,-42.615,178.771,5.889,149.416
C02464=1156.996,-109.258,-42.624,178.774,5.890,149.416
C02465=1156.991,-109.008,-42.633,178.775,5.890,149.415
C02466=1156.985,-108.758,-42.642,178.777,5.891,149.415
C02467=1156.980,-108.508,-42.651,178.780,5.890,149.414
C02468=1156.974,-108.259,-42.661,178.782,5.891,149.413
C02469=1156.969,-108.009,-42.669,178.784,5.892,149.413
C02470=1156.964,-107.759,-42.678,178.786,5.892,149.412
C02471=1156.959,-107.510,-42.687,178.788,5.892,149.412
C02472=1156.953,-107.259,-42.697,178.790,5.892,149.411
C02473=1156.948,-107.010,-42.706,178.792,5.893,149.411
C02474=1156.942,-106.760,-42.715,178.794,5.893,149.410
C02475=1156.937,-106.510,-42.723,178.796,5.893,149.410
C02476=1156.932,-106.260,-42.734,178.798,5.894,149.409
C02477=1156.926,-106.011,-42.743,178.800,5.894,149.409
C02478=1156.921,-105.761,-42.751,178.803,5.894,149.408
C02479=1156.916,-105.512,-42.760,178.804,5.894,149.407
C02480=1156.910,-105.262,-42.769,178.807,5.895,149.407
C02481=1156.904,-105.012,-42.778,178.808,5.895,149.406
C02482=1156.900,-104.762,-42.788,178.811,5.895,149.406
C02483=1156.894,-104.512,-42.797,178.813,5.896,149.405
C02484=1156.889,-104.262,-42.806,178.815,5.896,149.405
C02485=1156.883,-104.012,-42.815,178.817,5.896,149.404
C02486=1156.878,-103.763,-42.824,178.819,5.896,149.404
C02487=1156.873,-103.513,-42.834,178.821,5.897,149.403
C02488=1156.867,-103.263,-42.843,178.823,5.898,149.403
C02489=1156.862,-103.013,-42.852,178.825,5.897,149.402
C02490=1156.857,-102.741,-42.862,178.828,5.898,149.401
C02491=1156.851,-102.469,-42.873,178.830,5.899,149.401
C02492=1156.845,-102.198,-42.882,178.832,5.898,149.400
C02493=1156.839,-101.925,-42.893,178.834,5.899,149.399
C02494=1156.833,-101.676,-42.902,178.837,5.900,149.399
C02495=1156.829,-101.426,-42.911,178.838,5.900,149.398
C02496=1156.823,-101.176,-42.921,178.840,5.900,149.398
C02497=1156.818,-100.926,-42.930,178.843,5.900,149.397
C02498=1156.812,-100.676,-42.938,178.845,5.901,149.397
C02499=1156.807,-100.427,-42.949,178.847,5.901,149.396
C02500=1156.802,-100.177,-42.958,178.849,5.901,149.396
C02501=1156.796,-99.927,-42.966,178.851,5.902,149.395
C02502=1156.791,-99.678,-42.977,178.853,5.902,149.395
C02503=1156.786,-99.428,-42.986,178.855,5.902,149.394
C02504=1156.780,-99.178,-42.994,178.858,5.903,149.393
C02505=1156.775,-98.928,-43.005,178.859,5.903,149.393
C02506=1156.770,-98.679,-43.014,178.861,5.904,149.392
C02507=1156.764,-98.428,-43.023,178.864,5.903,149.392
C02508=1156.759,-98.179,-43.033,178.866,5.904,149.391
C02509=1156.754,-97.929,-43.042,178.868,5.905,149.391
C02510=1156.748,-97.679,-43.051,178.870,5.904,149.390
C02511=1156.743,-97.430,-43.061,178.872,5.905,149.390
C02512=1156.737,-97.180,-43.070,178.874,5.906,149.389
C02513=1156.732,-96.931,-43.080,178.876,5.905,149.388
C02514=1156.727,-96.681,-43.089,178.879,5.906,149.388
C02515=1156.721,-96.431,-43.098,178.880,5.906,149.387
C02516=1156.717,-96.181,-43.108,178.883,5.907,149.387
C02517=1156.711,-95.930,-43.118,178.885,5.907,149.386
C02518=1156.706,-95.681,-43.127,178.887,5.907,149.386
C02519=1156.700,-95.431,-43.137,178.889,5.908,149.385
C02520=1156.695,-95.182,-43.146,178.891,5.908,149.385
C02521=1156.690,-94.932,-43.156,178.893,5.908,149.384
C02522=1156.684,-94.682,-43.165,178.896,5.909,149.383
C02523=1156.679,-94.433,-43.174,178.897,5.909,149.383
C02524=1156.674,-94.182,-43.184,178.900,5.910,149.382
C02525=1156.669,-93.933,-43.193,178.902,5.910,149.382
C02526=1156.663,-93.683,-43.203,178.904,5.910,149.381
C02527=1156.658,-93.434,-43.213,178.906,5.911,149.381
C02528=1156.652,-93.184,-43.222,178.908,5.911,149.380
C02529=1156.647,-92.934,-43.232,178.910,5.911,149.379
C02530=1156.642,-92.683,-43.242,178.913,5.912,149.379
C02531=1156.637,-92.434,-43.251,178.914,5.912,149.379
C02532=1156.631,-92.184,-43.261,178.917,5.912,149.378
C02533=1156.626,-91.935,-43.270,178.919,5.913,149.377
C02534=1156.620,-91.685,-43.280,178.921,5.913,149.377
C02535=1156.615,-91.435,-43.289,178.923,5.913,149.376
C02536=1156.610,-91.186,-43.300,178.925,5.914,149.376
C02537=1156.605,-90.936,-43.308,178.927,5.914,149.375
C02538=1156.599,-90.687,-43.319,178.930,5.914,149.374
C02539=1156.594,-90.436,-43.329,178.932,5.915,149.374
C02540=1156.589,-90.186,-43.338,178.934,5.915,149.373
C02541=1156.583,-89.936,-43.348,178.936,5.915,149.373
C02542=1156.578,-89.687,-43.357,178.938,5.915,149.372
C02543=1156.573,-89.437,-43.367,178.940,5.916,149.372
C02544=1156.567,-89.188,-43.376,178.943,5.917,149.371
C02545=1156.562,-88.938,-43.387,178.944,5.917,149.371
C02546=1156.557,-88.688,-43.396,178.947,5.917,149.370
C02547=1156.552,-88.438,-43.406,178.949,5.918,149.369
C02548=1156.546,-88.188,-43.416,178.951,5.918,149.369
C02549=1156.541,-87.939,-43.425,178.953,5.918,149.368
C02550=1156.535,-87.689,-43.435,178.956,5.919,149.368
C02551=1156.530,-87.440,-43.445,178.957,5.919,149.367
C02552=1156.525,-87.189,-43.455,178.960,5.919,149.367
C02553=1156.520,-86.939,-43.465,178.962,5.920,149.366
C02554=1156.515,-86.690,-43.475,178.964,5.920,149.366
C02555=1156.509,-86.440,-43.484,178.966,5.920,149.365
C02556=1156.504,-86.191,-43.494,178.969,5.921,149.364
C02557=1156.498,-85.941,-43.504,178.970,5.921,149.364
C02558=1156.493,-85.690,-43.514,178.973,5.921,149.363
C02559=1156.488,-85.441,-43.523,178.975,5.922,149.363
C02560=1156.483,-85.192,-43.534,178.977,5.922,149.362
C02561=1156.477,-84.941,-43.543,178.979,5.923,149.361
C02562=1156.472,-84.692,-43.553,178.981,5.923,149.361
C02563=1156.467,-84.442,-43.563,178.984,5.923,149.360
C02564=1156.462,-84.193,-43.573,178.986,5.924,149.360
C02565=1156.456,-83.943,-43.582,178.988,5.925,149.359
C02566=1156.450,-83.693,-43.593,178.990,5.924,149.359
C02567=1156.446,-83.443,-43.603,178.992,5.925,149.358
C02568=1156.441,-83.194,-43.613,178.994,5.926,149.358
C02569=1156.435,-82.944,-43.623,178.996,5.925,149.357
C02570=1156.429,-82.694,-43.633,178.999,5.926,149.356
C02571=1156.424,-82.445,-43.642,179.001,5.927,149.356
C02572=1156.419,-82.194,-43.653,179.003,5.926,149.355
C02573=1156.414,-81.945,-43.663,179.005,5.927,149.355
C02574=1156.408,-81.695,-43.672,179.008,5.928,149.354
C02575=1156.403,-81.445,-43.682,179.010,5.928,149.354
C02576=1156.398,-81.195,-43.693,179.012,5.928,149.353
C02577=1156.392,-80.946,-43.703,179.014,5.929,149.352
C02578=1156.387,-80.696,-43.712,179.016,5.929,149.352
C02579=1156.382,-80.447,-43.723,179.018,5.929,149.351
C02580=1156.376,-80.196,-43.732,179.021,5.930,149.351
C02581=1156.371,-79.946,-43.743,179.023,5.931,149.350
C02582=1156.366,-79.697,-43.752,179.025,5.930,149.350
C02583=1156.361,-79.447,-43.763,179.027,5.931,149.349
C02584=1156.355,-79.197,-43.773,179.029,5.932,149.349
C02585=1156.350,-78.948,-43.783,179.031,5.931,149.348
C02586=1156.345,-78.699,-43.793,179.034,5.932,149.347
C02587=1156.340,-78.448,-43.803,179.036,5.933,149.347
C02588=1156.334,-78.199,-43.814,179.038,5.933,149.346
C02589=1156.328,-77.949,-43.823,179.040,5.933,149.346
C02590=1156.323,-77.698,-43.834,179.043,5.934,149.345
C02591=1156.319,-77.449,-43.843,179.045,5.934,149.345
C02592=1156.313,-77.200,-43.854,179.047,5.934,149.344
C02593=1156.307,-76.950,-43.864,179.049,5.935,149.343
C02594=1156.302,-76.679,-43.875,179.051,5.936,149.343
C02595=1156.296,-76.407,-43.886,179.054,5.936,149.342
C02596=1156.291,-76.137,-43.897,179.057,5.936,149.341
C02597=1156.285,-75.865,-43.908,179.058,5.936,149.341
C02598=1156.279,-75.616,-43.919,179.061,5.937,149.340
C02599=1156.274,-75.365,-43.929,179.063,5.937,149.340
C02600=1156.268,-75.116,-43.939,179.065,5.938,149.339
C02601=1156.264,-74.867,-43.949,179.067,5.938,149.339
C02602=1156.259,-74.616,-43.960,179.070,5.939,149.338
C02603=1156.253,-74.367,-43.970,179.072,5.939,149.337
C02604=1156.247,-74.117,-43.980,179.074,5.939,149.337
C02605=1156.242,-73.867,-43.991,179.076,5.940,149.336
C02606=1156.237,-73.617,-44.001,179.079,5.940,149.336
C02607=1156.231,-73.368,-44.011,179.081,5.941,149.335
C02608=1156.226,-73.118,-44.022,179.083,5.940,149.335
C02609=1156.221,-72.868,-44.031,179.085,5.941,149.334
C02610=1156.216,-72.618,-44.042,179.087,5.942,149.334
C02611=1156.211,-72.369,-44.052,179.090,5.942,149.333
C02612=1156.205,-72.119,-44.062,179.092,5.942,149.332
C02613=1156.200,-71.869,-44.073,179.094,5.943,149.332
C02614=1156.195,-71.619,-44.083,179.097,5.944,149.331
C02615=1156.189,-71.370,-44.094,179.098,5.944,149.331
C02616=1156.184,-71.120,-44.104,179.101,5.944,149.330
C02617=1156.179,-70.871,-44.115,179.103,5.945,149.330
C02618=1156.174,-70.620,-44.125,179.106,5.945,149.329
C02619=1156.168,-70.371,-44.135,179.107,5.945,149.328
C02620=1156.162,-70.121,-44.146,179.109,5.946,149.328
C02621=1156.157,-69.871,-44.156,179.112,5.946,149.327
C02622=1156.152,-69.621,-44.166,179.114,5.947,149.327
C02623=1156.147,-69.372,-44.178,179.116,5.947,149.326
C02624=1156.142,-69.122,-44.188,179.119,5.947,149.325
C02625=1156.136,-68.873,-44.198,179.121,5.948,149.325
C02626=1156.131,-68.622,-44.209,179.123,5.949,149.324
C02627=1156.125,-68.373,-44.219,179.125,5.949,149.324
C02628=1156.120,-68.123,-44.229,179.128,5.949,149.323
C02629=1156.115,-67.874,-44.240,179.130,5.950,149.323
C02630=1156.110,-67.623,-44.251,179.133,5.950,149.322
C02631=1156.104,-67.374,-44.261,179.134,5.950,149.321
C02632=1156.099,-67.124,-44.271,179.136,5.951,149.321
C02633=1156.094,-66.874,-44.282,179.139,5.951,149.320
C02634=1156.089,-66.625,-44.293,179.141,5.952,149.320
C02635=1156.084,-66.375,-44.303,179.143,5.952,149.319
C02636=1156.078,-66.125,-44.314,179.145,5.952,149.319
C02637=1156.073,-65.875,-44.324,179.148,5.953,149.318
C02638=1156.068,-65.626,-44.335,179.150,5.954,149.317
C02639=1156.063,-65.376,-44.346,179.152,5.954,149.317
C02640=1156.057,-65.126,-44.356,179.155,5.954,149.316
C02641=1156.052,-64.877,-44.367,179.157,5.955,149.316
C02642=1156.047,-64.627,-44.377,179.159,5.955,149.315
C02643=1156.042,-64.377,-44.388,179.162,5.956,149.315
C02644=1156.036,-64.128,-44.398,179.163,5.956,149.314
C02645=1156.032,-63.878,-44.410,179.166,5.956,149.313
C02646=1156.026,-63.628,-44.420,179.168,5.957,149.313
C02647=1156.021,-63.378,-44.430,179.171,5.958,149.312
C02648=1156.016,-63.129,-44.441,179.172,5.958,149.312
C02649=1156.010,-62.879,-44.452,179.175,5.958,149.311
C02650=1156.004,-62.629,-44.463,179.177,5.959,149.310
C02651=1156.000,-62.379,-44.474,179.179,5.960,149.310
C02652=1155.994,-62.130,-44.484,179.181,5.959,149.309
C02653=1155.989,-61.880,-44.495,179.184,5.960,149.309
C02654=1155.984,-61.631,-44.506,179.186,5.960,149.308
C02655=1155.979,-61.381,-44.516,179.189,5.961,149.308
C02656=1155.973,-61.132,-44.527,179.191,5.961,149.307
C02657=1155.968,-60.881,-44.538,179.193,5.961,149.306
C02658=1155.962,-60.632,-44.549,179.195,5.962,149.306
C02659=1155.957,-60.382,-44.560,179.198,5.963,149.305
C02660=1155.952,-60.132,-44.570,179.200,5.963,149.305
C02661=1155.947,-59.883,-44.581,179.202,5.964,149.304
C02662=1155.942,-59.632,-44.592,179.204,5.964,149.304
C02663=1155.937,-59.384,-44.603,179.207,5.964,149.303
C02664=1155.931,-59.133,-44.614,179.209,5.965,149.302
C02665=1155.926,-58.884,-44.625,179.212,5.965,149.302
C02666=1155.921,-58.634,-44.635,179.213,5.965,149.301
C02667=1155.916,-58.385,-44.646,179.215,5.966,149.301
C02668=1155.911,-58.135,-44.657,179.218,5.967,149.300
C02669=1155.906,-57.885,-44.668,179.220,5.967,149.300
C02670=1155.899,-57.635,-44.679,179.223,5.968,149.299
C02671=1155.895,-57.386,-44.690,179.224,5.968,149.298
C02672=1155.889,-57.136,-44.701,179.227,5.968,149.298
C02673=1155.884,-56.886,-44.712,179.229,5.969,149.297
C02674=1155.878,-56.637,-44.723,179.232,5.969,149.297
C02675=1155.873,-56.387,-44.734,179.234,5.970,149.296
C02676=1155.868,-56.137,-44.745,179.236,5.971,149.296
C02677=1155.863,-55.888,-44.755,179.238,5.971,149.295
C02678=1155.858,-55.637,-44.766,179.241,5.971,149.294
C02679=1155.853,-55.388,-44.778,179.243,5.972,149.294
C02680=1155.847,-55.139,-44.789,179.246,5.972,149.293
C02681=1155.842,-54.888,-44.799,179.248,5.973,149.292
C02682=1155.837,-54.639,-44.810,179.250,5.973,149.292
C02683=1155.831,-54.389,-44.821,179.252,5.973,149.291
C02684=1155.827,-54.139,-44.833,179.255,5.974,149.291
C02685=1155.821,-53.890,-44.843,179.257,5.975,149.290
C02686=1155.816,-53.640,-44.855,179.259,5.975,149.290
C02687=1155.811,-53.390,-44.866,179.262,5.976,149.289
C02688=1155.805,-53.141,-44.876,179.264,5.976,149.288
C02689=1155.801,-52.891,-44.888,179.266,5.976,149.288
C02690=1155.795,-52.641,-44.900,179.269,5.977,149.287
C02691=1155.790,-52.392,-44.910,179.271,5.978,149.287
C02692=1155.785,-52.142,-44.921,179.273,5.978,149.286
C02693=1155.780,-51.892,-44.933,179.275,5.978,149.286
C02694=1155.774,-51.642,-44.943,179.278,5.978,149.285
C02695=1155.769,-51.393,-44.954,179.280,5.979,149.284
C02696=1155.764,-51.143,-44.966,179.282,5.980,149.284
C02697=1155.758,-50.893,-44.977,179.285,5.980,149.283
C02698=1155.753,-50.623,-44.989,179.287,5.981,149.283
C02699=1155.747,-50.353,-45.001,179.290,5.982,149.282
C02700=1155.741,-50.082,-45.014,179.292,5.982,149.281
C02701=1155.735,-49.811,-45.026,179.295,5.982,149.281
C02702=1155.730,-49.562,-45.037,179.297,5.983,149.280
C02703=1155.725,-49.312,-45.047,179.299,5.983,149.279
C02704=1155.720,-49.062,-45.059,179.301,5.984,149.279
C02705=1155.715,-48.812,-45.071,179.304,5.984,149.279
C02706=1155.709,-48.563,-45.082,179.306,5.985,149.278
C02707=1155.704,-48.313,-45.093,179.308,5.986,149.277
C02708=1155.699,-48.063,-45.104,179.311,5.986,149.277
C02709=1155.693,-47.814,-45.115,179.313,5.987,149.276
C02710=1155.689,-47.564,-45.127,179.315,5.986,149.275
C02711=1155.683,-47.314,-45.139,179.318,5.987,149.275
C02712=1155.679,-47.064,-45.150,179.320,5.988,149.274
C02713=1155.672,-46.815,-45.161,179.322,5.988,149.274
C02714=1155.667,-46.565,-45.172,179.325,5.989,149.273
C02715=1155.663,-46.315,-45.183,179.327,5.990,149.273
C02716=1155.657,-46.065,-45.195,179.330,5.990,149.272
C02717=1155.652,-45.816,-45.206,179.331,5.990,149.271
C02718=1155.647,-45.567,-45.218,179.334,5.990,149.271
C02719=1155.642,-45.316,-45.229,179.336,5.991,149.270
C02720=1155.636,-45.066,-45.240,179.339,5.992,149.270
C02721=1155.631,-44.817,-45.251,179.341,5.992,149.269
C02722=1155.626,-44.567,-45.263,179.343,5.993,149.269
C02723=1155.621,-44.318,-45.275,179.346,5.994,149.268
C02724=1155.615,-44.068,-45.286,179.348,5.994,149.267
C02725=1155.610,-43.819,-45.297,179.350,5.994,149.267
C02726=1155.605,-43.569,-45.309,179.352,5.995,149.266
C02727=1155.600,-43.319,-45.321,179.355,5.995,149.266
C02728=1155.595,-43.070,-45.332,179.357,5.996,149.265
C02729=1155.590,-42.820,-45.344,179.360,5.996,149.264
C02730=1155.584,-42.570,-45.355,179.362,5.997,149.264
C02731=1155.579,-42.320,-45.366,179.365,5.998,149.263
C02732=1155.573,-42.070,-45.378,179.367,5.998,149.263
C02733=1155.569,-41.821,-45.389,179.369,5.998,149.262
C02734=1155.563,-41.571,-45.401,179.371,5.999,149.262
C02735=1155.557,-41.322,-45.412,179.374,5.999,149.261
C02736=1155.553,-41.072,-45.424,179.376,6.000,149.260
C02737=1155.547,-40.822,-45.436,179.379,6.000,149.260
C02738=1155.542,-40.572,-45.447,179.381,6.001,149.259
C02739=1155.537,-40.323,-45.459,179.383,6.002,149.259
C02740=1155.532,-40.073,-45.471,179.386,6.002,149.258
C02741=1155.526,-39.824,-45.482,179.388,6.003,149.258
C02742=1155.521,-39.574,-45.493,179.390,6.003,149.257
C02743=1155.516,-39.325,-45.505,179.392,6.004,149.256
C02744=1155.511,-39.075,-45.517,179.395,6.004,149.256
C02745=1155.506,-38.825,-45.529,179.397,6.005,149.255
C02746=1155.501,-38.575,-45.540,179.400,6.005,149.255
C02747=1155.495,-38.326,-45.552,179.402,6.006,149.254
C02748=1155.490,-38.076,-45.563,179.405,6.006,149.253
C02749=1155.485,-37.826,-45.575,179.407,6.007,149.253
C02750=1155.479,-37.577,-45.587,179.409,6.008,149.252
C02751=1155.475,-37.327,-45.598,179.412,6.008,149.252
C02752=1155.469,-37.077,-45.610,179.414,6.008,149.251
C02753=1155.464,-36.827,-45.622,179.416,6.009,149.251
C02754=1155.459,-36.578,-45.634,179.419,6.009,149.250
C02755=1155.453,-36.329,-45.646,179.421,6.010,149.249
C02756=1155.448,-36.079,-45.658,179.423,6.011,149.249
C02757=1155.443,-35.829,-45.669,179.426,6.011,149.248
C02758=1155.438,-35.579,-45.681,179.428,6.012,149.247
C02759=1155.432,-35.329,-45.693,179.430,6.013,149.247
C02760=1155.427,-35.080,-45.705,179.433,6.013,149.246
C02761=1155.423,-34.830,-45.716,179.435,6.014,149.246
C02762=1155.417,-34.580,-45.728,179.438,6.014,149.245
C02763=1155.412,-34.331,-45.740,179.440,6.015,149.245
C02764=1155.407,-34.081,-45.752,179.442,6.015,149.244
C02765=1155.402,-33.832,-45.764,179.444,6.015,149.243
C02766=1155.396,-33.582,-45.776,179.447,6.016,149.243
C02767=1155.390,-33.332,-45.788,179.449,6.017,149.242
C02768=1155.386,-33.083,-45.799,179.451,6.017,149.242
C02769=1155.381,-32.833,-45.811,179.454,6.018,149.241
C02770=1155.375,-32.584,-45.823,179.456,6.019,149.241
C02771=1155.370,-32.334,-45.835,179.459,6.019,149.240
C02772=1155.365,-32.084,-45.847,179.461,6.020,149.239
C02773=1155.360,-31.835,-45.859,179.464,6.020,149.239
C02774=1155.355,-31.585,-45.871,179.466,6.021,149.238
C02775=1155.349,-31.335,-45.883,179.469,6.021,149.238
C02776=1155.344,-31.085,-45.895,179.471,6.022,149.237
C02777=1155.339,-30.836,-45.907,179.473,6.023,149.236
C02778=1155.334,-30.586,-45.919,179.476,6.023,149.236
C02779=1155.328,-30.336,-45.931,179.478,6.024,149.235
C02780=1155.323,-30.087,-45.943,179.480,6.024,149.235
C02781=1155.318,-29.837,-45.955,179.483,6.024,149.234
C02782=1155.313,-29.588,-45.967,179.485,6.025,149.234
C02783=1155.308,-29.338,-45.979,179.487,6.026,149.233
C02784=1155.303,-29.088,-45.991,179.490,6.026,149.232
C02785=1155.297,-28.839,-46.003,179.492,6.027,149.232
C02786=1155.292,-28.589,-46.015,179.494,6.028,149.231
C02787=1155.287,-28.339,-46.027,179.497,6.028,149.231
C02788=1155.282,-28.090,-46.039,179.499,6.029,149.230
C02789=1155.277,-27.840,-46.051,179.502,6.029,149.229
C02790=1155.272,-27.590,-46.064,179.504,6.030,149.229
C02791=1155.266,-27.340,-46.076,179.507,6.030,149.228
C02792=1155.261,-27.091,-46.088,179.509,6.031,149.228
C02793=1155.256,-26.841,-46.100,179.512,6.032,149.227
C02794=1155.250,-26.591,-46.112,179.514,6.032,149.227
C02795=1155.245,-26.342,-46.125,179.516,6.033,149.226
C02796=1155.240,-26.092,-46.136,179.519,6.034,149.225
C02797=1155.235,-25.843,-46.148,179.521,6.034,149.225
C02798=1155.230,-25.593,-46.160,179.524,6.035,149.224
C02799=1155.225,-25.344,-46.173,179.526,6.035,149.224
C02800=1155.219,-25.094,-46.185,179.528,6.036,149.223
C02801=1155.215,-24.844,-46.198,179.531,6.037,149.222
C02802=1155.209,-24.574,-46.210,179.533,6.037,149.222
C02803=1155.204,-24.304,-46.224,179.536,6.038,149.221
C02804=1155.197,-24.034,-46.237,179.539,6.038,149.221
C02805=1155.192,-23.764,-46.250,179.541,6.039,149.220
C02806=1155.187,-23.515,-46.263,179.543,6.039,149.219
C02807=1155.181,-23.265,-46.275,179.546,6.040,149.219
C02808=1155.176,-23.016,-46.287,179.548,6.041,149.218
C02809=1155.171,-22.766,-46.300,179.550,6.041,149.218
C02810=1155.166,-22.516,-46.312,179.553,6.042,149.217
C02811=1155.161,-22.266,-46.325,179.555,6.043,149.217
C02812=1155.156,-22.016,-46.337,179.558,6.043,149.216
C02813=1155.151,-21.767,-46.349,179.560,6.044,149.215
C02814=1155.146,-21.518,-46.362,179.563,6.044,149.215
C02815=1155.140,-21.268,-46.374,179.565,6.045,149.214
C02816=1155.135,-21.018,-46.386,179.568,6.046,149.214
C02817=1155.130,-20.768,-46.398,179.570,6.046,149.213
C02818=1155.124,-20.519,-46.411,179.572,6.047,149.212
C02819=1155.120,-20.269,-46.424,179.575,6.048,149.212
C02820=1155.114,-20.019,-46.436,179.577,6.048,149.211
C02821=1155.109,-19.770,-46.448,179.579,6.049,149.211
C02822=1155.104,-19.521,-46.461,179.582,6.049,149.210
C02823=1155.099,-19.271,-46.473,179.584,6.050,149.210
C02824=1155.094,-19.021,-46.485,179.587,6.051,149.209
C02825=1155.089,-18.772,-46.498,179.589,6.051,149.208
C02826=1155.083,-18.522,-46.511,179.592,6.052,149.208
C02827=1155.078,-18.272,-46.523,179.594,6.053,149.207
C02828=1155.073,-18.022,-46.536,179.597,6.053,149.207
C02829=1155.068,-17.773,-46.549,179.599,6.054,149.206
C02830=1155.062,-17.523,-46.560,179.601,6.054,149.205
C02831=1155.057,-17.274,-46.573,179.604,6.055,149.205
C02832=1155.053,-17.024,-46.586,179.606,6.055,149.204
C02833=1155.047,-16.775,-46.599,179.608,6.056,149.204
C02834=1155.042,-16.525,-46.611,179.611,6.057,149.203
C02835=1155.037,-16.275,-46.623,179.613,6.058,149.203
C02836=1155.031,-16.026,-46.636,179.616,6.058,149.202
C02837=1155.026,-15.776,-46.649,179.618,6.059,149.201
C02838=1155.021,-15.526,-46.662,179.621,6.059,149.201
C02839=1155.016,-15.276,-46.674,179.624,6.061,149.200
C02840=1155.011,-15.027,-46.686,179.626,6.061,149.200
C02841=1155.006,-14.778,-46.699,179.628,6.062,149.199
C02842=1155.000,-14.527,-46.713,179.631,6.062,149.198
C02843=1154.995,-14.278,-46.725,179.633,6.063,149.198
C02844=1154.990,-14.029,-46.738,179.636,6.064,149.197
C02845=1154.985,-13.779,-46.750,179.638,6.064,149.197
C02846=1154.980,-13.529,-46.763,179.641,6.065,149.196
C02847=1154.975,-13.279,-46.775,179.643,6.066,149.196
C02848=1154.969,-13.030,-46.788,179.646,6.066,149.195
C02849=1154.964,-12.781,-46.801,179.648,6.067,149.194
C02850=1154.960,-12.531,-46.814,179.650,6.067,149.194
C02851=1154.954,-12.281,-46.827,179.653,6.068,149.193
C02852=1154.949,-12.032,-46.839,179.655,6.069,149.193
C02853=1154.943,-11.782,-46.852,179.657,6.069,149.192
C02854=1154.939,-11.532,-46.865,179.660,6.070,149.191
C02855=1154.934,-11.283,-46.878,179.662,6.071,149.191
C02856=1154.929,-11.034,-46.891,179.665,6.071,149.190
C02857=1154.923,-10.783,-46.904,179.667,6.072,149.190
C02858=1154.918,-10.534,-46.917,179.670,6.072,149.189
C02859=1154.913,-10.285,-46.929,179.672,6.073,149.188
C02860=1154.908,-10.035,-46.942,179.675,6.074,149.188
C02861=1154.903,-9.785,-46.955,179.678,6.075,149.187
C02862=1154.898,-9.536,-46.968,179.680,6.076,149.187
C02863=1154.893,-9.286,-46.981,179.683,6.076,149.186
C02864=1154.887,-9.036,-46.994,179.685,6.077,149.186
C02865=1154.882,-8.787,-47.007,179.688,6.077,149.185
C02866=1154.877,-8.537,-47.019,179.690,6.078,149.185
C02867=1154.873,-8.287,-47.032,179.692,6.079,149.184
C02868=1154.867,-8.038,-47.046,179.695,6.079,149.183
C02869=1154.862,-7.788,-47.058,179.697,6.080,149.183
C02870=1154.857,-7.538,-47.071,179.699,6.081,149.182
C02871=1154.851,-7.289,-47.084,179.702,6.081,149.182
C02872=1154.846,-7.039,-47.097,179.704,6.082,149.181
C02873=1154.842,-6.789,-47.110,179.707,6.082,149.180
C02874=1154.836,-6.540,-47.123,179.710,6.084,149.180
C02875=1154.831,-6.290,-47.136,179.712,6.084,149.179
C02876=1154.826,-6.041,-47.150,179.714,6.085,149.179
C02877=1154.820,-5.791,-47.163,179.717,6.086,149.178
C02878=1154.815,-5.542,-47.175,179.719,6.086,149.178
C02879=1154.810,-5.292,-47.189,179.722,6.087,149.177
C02880=1154.805,-5.042,-47.201,179.724,6.088,149.176
C02881=1154.800,-4.792,-47.214,179.727,6.088,149.176
C02882=1154.795,-4.543,-47.227,179.729,6.089,149.175
C02883=1154.790,-4.294,-47.241,179.732,6.089,149.175
C02884=1154.784,-4.044,-47.254,179.734,6.090,149.174
C02885=1154.779,-3.795,-47.267,179.737,6.091,149.173
C02886=1154.773,-3.545,-47.280,179.739,6.092,149.173
C02887=1154.769,-3.295,-47.293,179.742,6.093,149.172
C02888=1154.764,-3.046,-47.306,179.744,6.094,149.172
C02889=1154.759,-2.796,-47.320,179.747,6.094,149.171
C02890=1154.754,-2.547,-47.333,179.749,6.095,149.171
C02891=1154.749,-2.296,-47.346,179.752,6.095,149.170
C02892=1154.744,-2.047,-47.359,179.754,6.096,149.169
C02893=1154.738,-1.798,-47.373,179.756,6.097,149.169
C02894=1154.733,-1.548,-47.386,179.759,6.098,149.168
C02895=1154.727,-1.298,-47.399,179.762,6.099,149.168
C02896=1154.723,-1.049,-47.413,179.764,6.099,149.167
C02897=1154.717,-0.799,-47.426,179.767,6.100,149.166
C02898=1154.713,-0.549,-47.439,179.769,6.101,149.166
C02899=1154.707,-0.300,-47.453,179.771,6.101,149.165
C02900=1154.702,-0.051,-47.465,179.774,6.102,149.165
C02901=1154.697,0.200,-47.479,179.776,6.102,149.164
C02902=1154.692,0.448,-47.492,179.778,6.103,149.164
C02903=1154.687,0.699,-47.506,179.782,6.104,149.163
C02904=1154.682,0.948,-47.518,179.784,6.105,149.163
C02905=1154.677,1.198,-47.533,179.787,6.106,149.162
C02906=1154.670,1.467,-47.546,179.789,6.107,149.161
C02907=1154.666,1.736,-47.561,179.791,6.107,149.161
C02908=1154.660,2.006,-47.575,179.795,6.108,149.160
C02909=1154.655,2.275,-47.590,179.797,6.109,149.160
C02910=1154.649,2.525,-47.603,179.799,6.109,149.159
C02911=1154.644,2.774,-47.617,179.802,6.110,149.158
C02912=1154.639,3.024,-47.630,179.805,6.112,149.158
C02913=1154.634,3.274,-47.644,179.807,6.112,149.157
C02914=1154.629,3.523,-47.657,179.810,6.113,149.157
C02915=1154.624,3.773,-47.671,179.812,6.114,149.156
C02916=1154.618,4.022,-47.684,179.815,6.114,149.155
C02917=1154.613,4.272,-47.698,179.817,6.115,149.155
C02918=1154.608,4.521,-47.711,179.819,6.115,149.154
C02919=1154.603,4.771,-47.725,179.822,6.117,149.154
C02920=1154.598,5.020,-47.738,179.825,6.117,149.153
C02921=1154.593,5.270,-47.752,179.827,6.118,149.153
C02922=1154.587,5.520,-47.765,179.830,6.119,149.152
C02923=1154.583,5.769,-47.779,179.832,6.119,149.152
C02924=1154.578,6.019,-47.792,179.834,6.120,149.151
C02925=1154.572,6.268,-47.806,179.837,6.121,149.150
C02926=1154.568,6.518,-47.819,179.840,6.122,149.150
C02927=1154.562,6.767,-47.833,179.842,6.123,149.149
C02928=1154.557,7.018,-47.847,179.845,6.123,149.149
C02929=1154.552,7.266,-47.860,179.847,6.124,149.148
C02930=1154.547,7.516,-47.874,179.849,6.125,149.147
C02931=1154.542,7.766,-47.888,179.852,6.125,149.147
C02932=1154.537,8.015,-47.901,179.855,6.127,149.146
C02933=1154.532,8.265,-47.915,179.857,6.127,149.146
C02934=1154.526,8.514,-47.929,179.860,6.128,149.145
C02935=1154.521,8.764,-47.943,179.862,6.129,149.145
C02936=1154.516,9.013,-47.956,179.865,6.129,149.144
C02937=1154.511,9.263,-47.970,179.867,6.131,149.143
C02938=1154.506,9.513,-47.984,179.870,6.131,149.143
C02939=1154.501,9.763,-47.997,179.872,6.132,149.142
C02940=1154.496,10.012,-48.011,179.875,6.132,149.142
C02941=1154.491,10.262,-48.025,179.877,6.133,149.141
C02942=1154.486,10.511,-48.038,179.880,6.134,149.141
C02943=1154.481,10.761,-48.053,179.882,6.135,149.140
C02944=1154.476,11.010,-48.066,179.885,6.136,149.139
C02945=1154.471,11.260,-48.080,179.887,6.137,149.139
C02946=1154.466,11.510,-48.094,179.890,6.137,149.138
C02947=1154.460,11.759,-48.108,179.892,6.138,149.138
C02948=1154.455,12.008,-48.122,179.895,6.139,149.137
C02949=1154.451,12.258,-48.135,179.897,6.140,149.137
C02950=1154.445,12.507,-48.149,179.900,6.140,149.136
C02951=1154.440,12.757,-48.163,179.902,6.141,149.135
C02952=1154.435,13.007,-48.178,179.905,6.142,149.135
C02953=1154.429,13.256,-48.191,179.908,6.143,149.134
C02954=1154.425,13.506,-48.204,179.910,6.144,149.134
C02955=1154.420,13.756,-48.219,179.913,6.145,149.133
C02956=1154.414,14.005,-48.233,179.915,6.145,149.133
C02957=1154.410,14.254,-48.247,179.917,6.146,149.132
C02958=1154.404,14.505,-48.260,179.921,6.147,149.131
C02959=1154.399,14.754,-48.274,179.923,6.148,149.131
C02960=1154.394,15.003,-48.289,179.925,6.148,149.130
C02961=1154.389,15.253,-48.303,179.928,6.149,149.130
C02962=1154.384,15.502,-48.316,179.930,6.150,149.129
C02963=1154.379,15.751,-48.330,179.933,6.151,149.129
C02964=1154.374,16.001,-48.345,179.936,6.152,149.128
C02965=1154.369,16.252,-48.358,179.938,6.153,149.127
C02966=1154.363,16.501,-48.372,179.940,6.153,149.127
C02967=1154.358,16.750,-48.387,179.943,6.155,149.126
C02968=1154.353,17.000,-48.401,179.946,6.155,149.126
C02969=1154.348,17.250,-48.415,179.948,6.156,149.125
C02970=1154.343,17.499,-48.429,179.951,6.157,149.125
C02971=1154.338,17.748,-48.443,179.953,6.158,149.124
C02972=1154.333,17.998,-48.458,179.956,6.159,149.123
C02973=1154.328,18.248,-48.472,179.958,6.159,149.123
C02974=1154.322,18.497,-48.486,179.960,6.160,149.122
C02975=1154.317,18.747,-48.500,179.963,6.161,149.122
C02976=1154.313,18.996,-48.514,179.966,6.162,149.121
C02977=1154.308,19.246,-48.528,179.968,6.163,149.121
C02978=1154.303,19.495,-48.542,179.971,6.164,149.120
C02979=1154.298,19.744,-48.556,179.973,6.164,149.120
C02980=1154.293,19.994,-48.570,179.976,6.166,149.119
C02981=1154.288,20.244,-48.585,179.979,6.166,149.118
C02982=1154.282,20.493,-48.599,179.981,6.167,149.118
C02983=1154.277,20.743,-48.613,179.984,6.167,149.117
C02984=1154.272,20.993,-48.628,179.986,6.169,149.117
C02985=1154.267,21.242,-48.642,179.989,6.170,149.116
C02986=1154.262,21.492,-48.656,179.991,6.170,149.116
C02987=1154.256,21.741,-48.670,179.994,6.171,149.115
C02988=1154.251,21.991,-48.685,179.997,6.172,149.115
C02989=1154.246,22.240,-48.699,179.999,6.173,149.114
C02990=1154.242,22.489,-48.714,-179.999,6.174,149.113
C02991=1154.237,22.739,-48.728,-179.996,6.174,149.113
C02992=1154.232,22.989,-48.742,-179.993,6.176,149.112
C02993=1154.226,23.238,-48.756,-179.991,6.176,149.112
C02994=1154.221,23.488,-48.771,-179.988,6.177,149.111
C02995=1154.216,23.737,-48.785,-179.985,6.178,149.110
C02996=1154.211,23.987,-48.799,-179.983,6.179,149.110
C02997=1154.207,24.236,-48.814,-179.980,6.180,149.109
C02998=1154.201,24.486,-48.829,-179.978,6.181,149.109
C02999=1154.196,24.736,-48.843,-179.975,6.182,149.108
C03000=1154.190,24.985,-48.857,-179.973,6.183,149.108
C03001=1154.185,25.235,-48.871,-179.971,6.183,149.107
C03002=1154.181,25.484,-48.886,-179.968,6.184,149.107
C03003=1154.176,25.733,-48.901,-179.965,6.186,149.106
C03004=1154.171,25.983,-48.915,-179.963,6.186,149.105
C03005=1154.166,26.233,-48.929,-179.960,6.187,149.105
C03006=1154.160,26.483,-48.944,-179.957,6.188,149.104
C03007=1154.156,26.732,-48.959,-179.955,6.189,149.104
C03008=1154.150,26.981,-48.973,-179.952,6.189,149.103
C03009=1154.145,27.231,-48.987,-179.950,6.191,149.103
C03010=1154.140,27.499,-49.003,-179.947,6.192,149.102
C03011=1154.134,27.769,-49.019,-179.944,6.192,149.101
C03012=1154.129,28.037,-49.035,-179.942,6.194,149.101
C03013=1154.124,28.306,-49.051,-179.939,6.194,149.100
C03014=1154.118,28.556,-49.066,-179.936,6.196,149.100
C03015=1154.113,28.806,-49.080,-179.933,6.196,149.099
C03016=1154.109,29.055,-49.095,-179.931,6.197,149.099
C03017=1154.104,29.305,-49.109,-179.928,6.198,149.098
C03018=1154.098,29.555,-49.124,-179.926,6.199,149.098
C03019=1154.093,29.804,-49.139,-179.923,6.200,149.097
C03020=1154.088,30.053,-49.153,-179.921,6.201,149.096
C03021=1154.083,30.302,-49.167,-179.918,6.202,149.096
C03022=1154.077,30.552,-49.183,-179.916,6.203,149.095
C03023=1154.072,30.802,-49.197,-179.913,6.203,149.095
C03024=1154.068,31.051,-49.212,-179.910,6.205,149.094
C03025=1154.063,31.300,-49.226,-179.908,6.205,149.093
C03026=1154.057,31.550,-49.242,-179.905,6.206,149.093
C03027=1154.052,31.800,-49.256,-179.903,6.208,149.093
C03028=1154.048,32.049,-49.270,-179.900,6.208,149.092
C03029=1154.042,32.299,-49.286,-179.898,6.209,149.091
C03030=1154.037,32.548,-49.300,-179.895,6.210,149.091
C03031=1154.033,32.797,-49.315,-179.893,6.211,149.090
C03032=1154.027,33.047,-49.330,-179.890,6.211,149.090
C03033=1154.022,33.297,-49.345,-179.887,6.213,149.089
C03034=1154.017,33.546,-49.359,-179.884,6.214,149.089
C03035=1154.012,33.796,-49.375,-179.882,6.214,149.088
C03036=1154.007,34.045,-49.389,-179.879,6.216,149.087
C03037=1154.002,34.294,-49.404,-179.877,6.217,149.087
C03038=1153.997,34.544,-49.419,-179.874,6.217,149.086
C03039=1153.992,34.794,-49.434,-179.872,6.219,149.086
C03040=1153.987,35.043,-49.449,-179.869,6.220,149.085
C03041=1153.982,35.293,-49.464,-179.867,6.220,149.085
C03042=1153.977,35.542,-49.479,-179.864,6.222,149.084
C03043=1153.972,35.792,-49.494,-179.861,6.222,149.084
C03044=1153.967,36.042,-49.509,-179.859,6.223,149.083
C03045=1153.963,36.291,-49.524,-179.856,6.224,149.082
C03046=1153.957,36.541,-49.539,-179.854,6.225,149.082
C03047=1153.952,36.790,-49.554,-179.851,6.226,149.081
C03048=1153.946,37.040,-49.569,-179.848,6.227,149.081
C03049=1153.942,37.289,-49.584,-179.846,6.228,149.080
C03050=1153.936,37.538,-49.600,-179.843,6.229,149.080
C03051=1153.932,37.788,-49.614,-179.841,6.230,149.079
C03052=1153.926,38.037,-49.629,-179.838,6.231,149.079
C03053=1153.921,38.286,-49.644,-179.835,6.232,149.078
C03054=1153.916,38.537,-49.659,-179.833,6.233,149.077
C03055=1153.911,38.786,-49.674,-179.831,6.234,149.077
C03056=1153.906,39.035,-49.690,-179.827,6.235,149.076
C03057=1153.902,39.285,-49.705,-179.825,6.236,149.076
C03058=1153.896,39.535,-49.720,-179.822,6.237,149.075
C03059=1153.891,39.784,-49.735,-179.820,6.238,149.075
C03060=1153.886,40.033,-49.751,-179.817,6.238,149.074
C03061=1153.881,40.282,-49.766,-179.814,6.240,149.074
C03062=1153.876,40.532,-49.781,-179.812,6.241,149.073
C03063=1153.871,40.782,-49.796,-179.810,6.241,149.073
C03064=1153.866,41.031,-49.811,-179.807,6.243,149.072
C03065=1153.862,41.281,-49.827,-179.804,6.243,149.071
C03066=1153.856,41.531,-49.841,-179.801,6.245,149.071
C03067=1153.851,41.780,-49.856,-179.799,6.245,149.070
C03068=1153.846,42.029,-49.872,-179.797,6.246,149.070
C03069=1153.841,42.278,-49.887,-179.793,6.248,149.069
C03070=1153.836,42.528,-49.903,-179.791,6.248,149.069
C03071=1153.830,42.777,-49.918,-179.788,6.250,149.068
C03072=1153.826,43.027,-49.933,-179.786,6.251,149.068
C03073=1153.821,43.277,-49.948,-179.784,6.251,149.067
C03074=1153.816,43.526,-49.963,-179.780,6.253,149.067
C03075=1153.811,43.775,-49.979,-179.778,6.254,149.066
C03076=1153.805,44.025,-49.995,-179.775,6.255,149.065
C03077=1153.801,44.275,-50.010,-179.773,6.256,149.065
C03078=1153.796,44.524,-50.025,-179.771,6.257,149.065
C03079=1153.791,44.773,-50.040,-179.768,6.258,149.064
C03080=1153.786,45.023,-50.056,-179.765,6.259,149.063
C03081=1153.780,45.272,-50.072,-179.762,6.260,149.063
C03082=1153.776,45.522,-50.087,-179.760,6.261,149.062
C03083=1153.771,45.771,-50.103,-179.757,6.261,149.062
C03084=1153.766,46.021,-50.118,-179.755,6.263,149.061
C03085=1153.761,46.270,-50.133,-179.752,6.263,149.060
C03086=1153.756,46.519,-50.149,-179.749,6.265,149.060
C03087=1153.751,46.769,-50.165,-179.747,6.266,149.060
C03088=1153.746,47.018,-50.180,-179.744,6.267,149.059
C03089=1153.741,47.268,-50.195,-179.742,6.268,149.058
C03090=1153.735,47.517,-50.211,-179.739,6.269,149.058
C03091=1153.731,47.767,-50.227,-179.736,6.270,149.057
C03092=1153.726,48.016,-50.242,-179.734,6.271,149.057
C03093=1153.720,48.266,-50.257,-179.731,6.272,149.056
C03094=1153.716,48.516,-50.273,-179.729,6.273,149.056
C03095=1153.711,48.765,-50.288,-179.725,6.274,149.055
C03096=1153.706,49.014,-50.304,-179.723,6.275,149.055
C03097=1153.700,49.264,-50.320,-179.721,6.276,149.054
C03098=1153.695,49.514,-50.335,-179.718,6.277,149.054
C03099=1153.691,49.763,-50.350,-179.715,6.278,149.053
C03100=1153.685,50.012,-50.366,-179.713,6.280,149.052
C03101=1153.681,50.262,-50.383,-179.710,6.280,149.052
C03102=1153.676,50.511,-50.398,-179.707,6.282,149.051
C03103=1153.670,50.761,-50.414,-179.705,6.283,149.051
C03104=1153.666,51.010,-50.429,-179.702,6.283,149.050
C03105=1153.661,51.260,-50.445,-179.700,6.285,149.050
C03106=1153.655,51.509,-50.460,-179.697,6.286,149.049
C03107=1153.650,51.758,-50.477,-179.694,6.287,149.049
C03108=1153.646,52.008,-50.493,-179.692,6.288,149.048
C03109=1153.641,52.257,-50.508,-179.689,6.289,149.048
C03110=1153.635,52.506,-50.523,-179.687,6.290,149.047
C03111=1153.631,52.757,-50.539,-179.683,6.291,149.046
C03112=1153.626,53.005,-50.556,-179.681,6.292,149.046
C03113=1153.620,53.255,-50.571,-179.679,6.294,149.046
C03114=1153.615,53.524,-50.589,-179.676,6.294,149.045
C03115=1153.610,53.792,-50.606,-179.673,6.295,149.044
C03116=1153.604,54.061,-50.623,-179.670,6.297,149.044
C03117=1153.599,54.329,-50.640,-179.667,6.298,149.043
C03118=1153.595,54.579,-50.655,-179.664,6.299,149.043
C03119=1153.589,54.828,-50.671,-179.662,6.300,149.042
C03120=1153.584,55.077,-50.687,-179.659,6.301,149.042
C03121=1153.579,55.327,-50.703,-179.657,6.302,149.041
C03122=1153.574,55.576,-50.719,-179.654,6.303,149.041
C03123=1153.569,55.826,-50.735,-179.652,6.304,149.040
C03124=1153.564,56.076,-50.751,-179.648,6.306,149.039
C03125=1153.559,56.325,-50.767,-179.646,6.306,149.039
C03126=1153.554,56.575,-50.783,-179.643,6.308,149.039
C03127=1153.549,56.824,-50.798,-179.641,6.309,149.038
C03128=1153.544,57.074,-50.815,-179.638,6.310,149.037
C03129=1153.539,57.323,-50.831,-179.635,6.311,149.037
C03130=1153.534,57.572,-50.847,-179.633,6.312,149.036
C03131=1153.529,57.822,-50.863,-179.631,6.313,149.036
C03132=1153.524,58.071,-50.879,-179.627,6.315,149.035
C03133=1153.519,58.321,-50.895,-179.625,6.315,149.035
C03134=1153.514,58.570,-50.911,-179.622,6.317,149.034
C03135=1153.509,58.820,-50.927,-179.620,6.318,149.034
C03136=1153.504,59.069,-50.943,-179.617,6.319,149.033
C03137=1153.499,59.318,-50.959,-179.614,6.320,149.033
C03138=1153.494,59.568,-50.975,-179.612,6.321,149.032
C03139=1153.489,59.817,-50.992,-179.609,6.322,149.031
C03140=1153.484,60.067,-51.008,-179.606,6.324,149.031
C03141=1153.479,60.316,-51.024,-179.604,6.324,149.031
C03142=1153.474,60.566,-51.040,-179.601,6.326,149.030
C03143=1153.469,60.814,-51.056,-179.599,6.327,149.030
C03144=1153.464,61.065,-51.072,-179.595,6.328,149.029
C03145=1153.459,61.313,-51.088,-179.593,6.329,149.028
C03146=1153.455,61.563,-51.105,-179.591,6.330,149.028
C03147=1153.450,61.812,-51.121,-179.588,6.331,149.027
C03148=1153.445,62.062,-51.137,-179.585,6.332,149.027
C03149=1153.439,62.311,-51.154,-179.583,6.333,149.026
C03150=1153.434,62.561,-51.170,-179.580,6.335,149.026
C03151=1153.429,62.810,-51.186,-179.578,6.336,149.025
C03152=1153.425,63.060,-51.202,-179.574,6.337,149.025
C03153=1153.419,63.309,-51.219,-179.572,6.338,149.024
C03154=1153.415,63.559,-51.235,-179.570,6.339,149.024
C03155=1153.410,63.807,-51.251,-179.567,6.340,149.023
C03156=1153.405,64.057,-51.268,-179.564,6.341,149.023
C03157=1153.400,64.307,-51.284,-179.561,6.343,149.022
C03158=1153.395,64.556,-51.301,-179.559,6.344,149.022
C03159=1153.390,64.806,-51.317,-179.556,6.345,149.021
C03160=1153.385,65.054,-51.333,-179.553,6.346,149.021
C03161=1153.380,65.305,-51.349,-179.551,6.347,149.020
C03162=1153.375,65.553,-51.366,-179.549,6.348,149.020
C03163=1153.370,65.803,-51.383,-179.545,6.350,149.019
C03164=1153.365,66.053,-51.399,-179.543,6.350,149.019
C03165=1153.360,66.302,-51.415,-179.540,6.352,149.018
C03166=1153.356,66.551,-51.432,-179.538,6.353,149.017
C03167=1153.350,66.800,-51.448,-179.535,6.354,149.017
C03168=1153.345,67.050,-51.466,-179.532,6.356,149.016
C03169=1153.340,67.300,-51.481,-179.530,6.356,149.016
C03170=1153.335,67.549,-51.498,-179.527,6.358,149.015
C03171=1153.331,67.798,-51.514,-179.524,6.359,149.015
C03172=1153.325,68.047,-51.531,-179.522,6.360,149.014
C03173=1153.321,68.297,-51.548,-179.519,6.361,149.014
C03174=1153.316,68.547,-51.564,-179.516,6.362,149.013
C03175=1153.311,68.796,-51.580,-179.513,6.364,149.013
C03176=1153.305,69.046,-51.598,-179.511,6.365,149.012
C03177=1153.301,69.295,-51.614,-179.508,6.366,149.012
C03178=1153.296,69.544,-51.631,-179.506,6.367,149.011
C03179=1153.291,69.794,-51.648,-179.503,6.368,149.011
C03180=1153.286,70.043,-51.664,-179.501,6.369,149.010
C03181=1153.281,70.292,-51.681,-179.498,6.371,149.010
C03182=1153.276,70.542,-51.698,-179.495,6.372,149.009
C03183=1153.271,70.791,-51.714,-179.492,6.373,149.009
C03184=1153.266,71.041,-51.730,-179.490,6.375,149.008
C03185=1153.261,71.290,-51.748,-179.487,6.375,149.008
C03186=1153.256,71.539,-51.764,-179.484,6.377,149.007
C03187=1153.251,71.789,-51.780,-179.482,6.379,149.007
C03188=1153.246,72.039,-51.798,-179.479,6.379,149.006
C03189=1153.241,72.287,-51.814,-179.476,6.381,149.006
C03190=1153.237,72.537,-51.831,-179.474,6.382,149.005
C03191=1153.231,72.787,-51.848,-179.471,6.383,149.005
C03192=1153.227,73.036,-51.865,-179.469,6.384,149.004
C03193=1153.221,73.285,-51.882,-179.465,6.385,149.004
C03194=1153.217,73.535,-51.898,-179.463,6.387,149.003
C03195=1153.212,73.784,-51.915,-179.461,6.388,149.003
C03196=1153.206,74.033,-51.932,-179.457,6.389,149.002
C03197=1153.202,74.282,-51.949,-179.455,6.391,149.002
C03198=1153.197,74.532,-51.966,-179.452,6.392,149.001
C03199=1153.192,74.781,-51.983,-179.449,6.393,149.000
C03200=1153.187,75.030,-52.000,-179.447,6.394,149.000
C03201=1153.182,75.280,-52.017,-179.444,6.395,149.000
C03202=1153.177,75.530,-52.034,-179.441,6.397,148.999
C03203=1153.172,75.779,-52.051,-179.439,6.398,148.999
C03204=1153.167,76.028,-52.067,-179.436,6.399,148.998
C03205=1153.162,76.278,-52.084,-179.434,6.400,148.997
C03206=1153.158,76.527,-52.102,-179.431,6.401,148.997
C03207=1153.153,76.776,-52.119,-179.428,6.403,148.997
C03208=1153.148,77.025,-52.135,-179.425,6.404,148.996
C03209=1153.142,77.275,-52.152,-179.423,6.405,148.996
C03210=1153.138,77.525,-52.169,-179.420,6.407,148.995
C03211=1153.133,77.774,-52.187,-179.417,6.407,148.994
C03212=1153.128,78.024,-52.204,-179.415,6.409,148.994
C03213=1153.123,78.272,-52.221,-179.412,6.411,148.994
C03214=1153.117,78.522,-52.238,-179.409,6.411,148.993
C03215=1153.113,78.771,-52.255,-179.407,6.413,148.992
C03216=1153.108,79.021,-52.273,-179.404,6.414,148.992
C03217=1153.104,79.270,-52.289,-179.401,6.415,148.991
C03218=1153.098,79.538,-52.308,-179.398,6.417,148.991
C03219=1153.092,79.807,-52.326,-179.396,6.419,148.991
C03220=1153.088,80.075,-52.345,-179.392,6.420,148.990
C03221=1153.082,80.343,-52.363,-179.390,6.421,148.989
C03222=1153.077,80.593,-52.381,-179.387,6.422,148.989
C03223=1153.072,80.843,-52.397,-179.384,6.424,148.988
C03224=1153.067,81.092,-52.415,-179.382,6.425,148.988
C03225=1153.063,81.341,-52.432,-179.379,6.426,148.987
C03226=1153.057,81.590,-52.449,-179.376,6.428,148.987
C03227=1153.052,81.840,-52.467,-179.374,6.428,148.986
C03228=1153.048,82.089,-52.483,-179.371,6.430,148.986
C03229=1153.043,82.338,-52.501,-179.368,6.431,148.985
C03230=1153.037,82.588,-52.519,-179.366,6.432,148.985
C03231=1153.033,82.838,-52.535,-179.363,6.434,148.984
C03232=1153.028,83.087,-52.553,-179.360,6.435,148.984
C03233=1153.023,83.337,-52.571,-179.358,6.436,148.983
C03234=1153.018,83.585,-52.588,-179.355,6.437,148.983
C03235=1153.013,83.834,-52.605,-179.352,6.439,148.982
C03236=1153.008,84.084,-52.623,-179.350,6.440,148.982
C03237=1153.003,84.333,-52.640,-179.347,6.442,148.982
C03238=1152.999,84.582,-52.658,-179.344,6.443,148.981
C03239=1152.993,84.832,-52.675,-179.341,6.445,148.980
C03240=1152.988,85.081,-52.693,-179.339,6.446,148.980
C03241=1152.984,85.331,-52.709,-179.336,6.447,148.979
C03242=1152.979,85.580,-52.727,-179.333,6.449,148.979
C03243=1152.974,85.830,-52.745,-179.331,6.449,148.979
C03244=1152.969,86.079,-52.763,-179.328,6.451,148.978
C03245=1152.964,86.328,-52.779,-179.325,6.452,148.977
C03246=1152.959,86.578,-52.797,-179.323,6.453,148.977
C03247=1152.954,86.827,-52.814,-179.320,6.455,148.977
C03248=1152.949,87.076,-52.832,-179.317,6.456,148.976
C03249=1152.944,87.325,-52.850,-179.315,6.457,148.976
C03250=1152.939,87.574,-52.867,-179.312,6.459,148.975
C03251=1152.934,87.824,-52.885,-179.309,6.461,148.975
C03252=1152.930,88.073,-52.903,-179.306,6.462,148.974
C03253=1152.924,88.323,-52.920,-179.304,6.463,148.974
C03254=1152.919,88.572,-52.938,-179.301,6.464,148.973
C03255=1152.915,88.821,-52.955,-179.298,6.466,148.973
C03256=1152.910,89.070,-52.973,-179.296,6.467,148.972
C03257=1152.905,89.320,-52.991,-179.293,6.468,148.972
C03258=1152.900,89.569,-53.009,-179.290,6.470,148.971
C03259=1152.895,89.819,-53.026,-179.287,6.471,148.971
C03260=1152.890,90.068,-53.044,-179.285,6.472,148.970
C03261=1152.885,90.317,-53.062,-179.282,6.474,148.970
C03262=1152.881,90.566,-53.079,-179.279,6.475,148.969
C03263=1152.876,90.816,-53.097,-179.277,6.476,148.969
C03264=1152.871,91.065,-53.115,-179.274,6.478,148.968
C03265=1152.866,91.314,-53.133,-179.271,6.479,148.968
C03266=1152.861,91.564,-53.150,-179.268,6.481,148.967
C03267=1152.856,91.814,-53.168,-179.266,6.482,148.967
C03268=1152.851,92.063,-53.186,-179.263,6.483,148.966
C03269=1152.847,92.312,-53.204,-179.261,6.485,148.966
C03270=1152.842,92.561,-53.222,-179.257,6.486,148.965
C03271=1152.836,92.811,-53.239,-179.255,6.487,148.965
C03272=1152.832,93.060,-53.257,-179.253,6.489,148.965
C03273=1152.827,93.309,-53.275,-179.250,6.491,148.964
C03274=1152.822,93.558,-53.293,-179.247,6.492,148.963
C03275=1152.817,93.808,-53.311,-179.244,6.493,148.963
C03276=1152.812,94.057,-53.329,-179.242,6.494,148.963
C03277=1152.807,94.306,-53.347,-179.239,6.496,148.962
C03278=1152.802,94.555,-53.365,-179.236,6.497,148.962
C03279=1152.797,94.805,-53.382,-179.234,6.498,148.961
C03280=1152.793,95.055,-53.401,-179.231,6.500,148.961
C03281=1152.788,95.304,-53.419,-179.228,6.502,148.960
C03282=1152.783,95.553,-53.437,-179.225,6.503,148.960
C03283=1152.778,95.802,-53.455,-179.223,6.504,148.959
C03284=1152.773,96.052,-53.473,-179.220,6.506,148.959
C03285=1152.768,96.301,-53.491,-179.217,6.507,148.958
C03286=1152.763,96.550,-53.509,-179.214,6.509,148.958
C03287=1152.758,96.799,-53.527,-179.212,6.510,148.957
C03288=1152.754,97.049,-53.545,-179.209,6.511,148.957
C03289=1152.749,97.298,-53.563,-179.207,6.513,148.957
C03290=1152.744,97.547,-53.581,-179.203,6.514,148.956
C03291=1152.739,97.797,-53.599,-179.201,6.516,148.955
C03292=1152.734,98.046,-53.617,-179.198,6.517,148.955
C03293=1152.729,98.295,-53.635,-179.196,6.518,148.955
C03294=1152.724,98.545,-53.654,-179.193,6.520,148.954
C03295=1152.719,98.794,-53.672,-179.190,6.521,148.954
C03296=1152.714,99.043,-53.690,-179.188,6.522,148.953
C03297=1152.710,99.292,-53.709,-179.185,6.524,148.953
C03298=1152.705,99.541,-53.726,-179.182,6.525,148.952
C03299=1152.701,99.791,-53.745,-179.179,6.527,148.952
C03300=1152.696,100.040,-53.763,-179.176,6.529,148.951
C03301=1152.690,100.290,-53.781,-179.174,6.530,148.951
C03302=1152.685,100.539,-53.799,-179.171,6.531,148.950
C03303=1152.680,100.788,-53.817,-179.168,6.533,148.950
C03304=1152.676,101.037,-53.836,-179.165,6.534,148.949
C03305=1152.671,101.286,-53.854,-179.163,6.536,148.949
C03306=1152.666,101.536,-53.872,-179.161,6.537,148.949
C03307=1152.661,101.785,-53.891,-179.157,6.538,148.948
C03308=1152.656,102.034,-53.909,-179.155,6.540,148.948
C03309=1152.652,102.284,-53.928,-179.152,6.542,148.947
C03310=1152.647,102.533,-53.946,-179.149,6.543,148.947
C03311=1152.641,102.782,-53.965,-179.147,6.544,148.946
C03312=1152.636,103.031,-53.983,-179.144,6.546,148.946
C03313=1152.632,103.281,-54.002,-179.141,6.547,148.945
C03314=1152.627,103.530,-54.020,-179.138,6.549,148.945
C03315=1152.622,103.779,-54.038,-179.136,6.551,148.944
C03316=1152.617,104.029,-54.056,-179.133,6.552,148.944
C03317=1152.613,104.278,-54.075,-179.130,6.553,148.943
C03318=1152.608,104.527,-54.093,-179.128,6.555,148.943
C03319=1152.602,104.776,-54.112,-179.125,6.556,148.943
C03320=1152.598,105.026,-54.131,-179.122,6.558,148.942
C03321=1152.593,105.275,-54.149,-179.119,6.560,148.942
C03322=1152.588,105.543,-54.169,-179.116,6.561,148.941
C03323=1152.583,105.811,-54.189,-179.113,6.563,148.941
C03324=1152.578,106.080,-54.209,-179.110,6.564,148.940
C03325=1152.572,106.349,-54.229,-179.108,6.566,148.940
C03326=1152.567,106.597,-54.248,-179.105,6.567,148.939
C03327=1152.563,106.847,-54.266,-179.102,6.569,148.939
C03328=1152.558,107.096,-54.284,-179.100,6.570,148.938
C03329=1152.553,107.345,-54.304,-179.097,6.571,148.938
C03330=1152.548,107.595,-54.322,-179.094,6.573,148.937
C03331=1152.543,107.844,-54.341,-179.091,6.575,148.937
C03332=1152.538,108.093,-54.359,-179.089,6.576,148.937
C03333=1152.534,108.343,-54.378,-179.086,6.578,148.936
C03334=1152.528,108.592,-54.397,-179.083,6.579,148.935
C03335=1152.524,108.841,-54.416,-179.081,6.580,148.935
C03336=1152.519,109.091,-54.434,-179.078,6.582,148.935
C03337=1152.514,109.339,-54.453,-179.075,6.584,148.934
C03338=1152.510,109.589,-54.472,-179.072,6.585,148.934
C03339=1152.504,109.838,-54.491,-179.070,6.587,148.933
C03340=1152.500,110.087,-54.509,-179.066,6.588,148.933
C03341=1152.495,110.337,-54.528,-179.064,6.590,148.932
C03342=1152.490,110.586,-54.546,-179.062,6.591,148.932
C03343=1152.485,110.835,-54.566,-179.059,6.593,148.932
C03344=1152.481,111.084,-54.585,-179.056,6.594,148.931
C03345=1152.475,111.334,-54.603,-179.053,6.596,148.931
C03346=1152.471,111.583,-54.622,-179.050,6.597,148.930
C03347=1152.465,111.832,-54.641,-179.047,6.599,148.930
C03348=1152.461,112.082,-54.660,-179.045,6.601,148.929
C03349=1152.456,112.330,-54.679,-179.042,6.603,148.929
C03350=1152.451,112.580,-54.697,-179.039,6.604,148.928
C03351=1152.446,112.829,-54.717,-179.037,6.605,148.928
C03352=1152.442,113.078,-54.736,-179.034,6.606,148.927
C03353=1152.437,113.328,-54.755,-179.031,6.608,148.927
C03354=1152.432,113.576,-54.773,-179.029,6.610,148.927
C03355=1152.427,113.826,-54.793,-179.026,6.612,148.926
C03356=1152.422,114.075,-54.812,-179.023,6.613,148.926
C03357=1152.418,114.325,-54.831,-179.020,6.615,148.925
C03358=1152.412,114.574,-54.850,-179.018,6.617,148.925
C03359=1152.408,114.823,-54.869,-179.014,6.618,148.924
C03360=1152.403,115.072,-54.888,-179.012,6.619,148.924
C03361=1152.398,115.322,-54.907,-179.010,6.621,148.924
C03362=1152.393,115.571,-54.926,-179.007,6.622,148.923
C03363=1152.388,115.820,-54.946,-179.004,6.624,148.923
C03364=1152.384,116.069,-54.964,-179.001,6.626,148.922
C03365=1152.379,116.318,-54.984,-178.999,6.627,148.922
C03366=1152.373,116.568,-55.002,-178.996,6.629,148.921
C03367=1152.369,116.817,-55.022,-178.993,6.630,148.921
C03368=1152.364,117.066,-55.041,-178.990,6.632,148.921
C03369=1152.359,117.315,-55.060,-178.987,6.634,148.920
C03370=1152.355,117.564,-55.079,-178.985,6.636,148.920
C03371=1152.350,117.814,-55.099,-178.982,6.637,148.919
C03372=1152.345,118.062,-55.118,-178.980,6.638,148.919
C03373=1152.341,118.312,-55.137,-178.977,6.640,148.918
C03374=1152.335,118.561,-55.156,-178.974,6.641,148.918
C03375=1152.330,118.811,-55.175,-178.971,6.643,148.917
C03376=1152.325,119.060,-55.195,-178.968,6.645,148.917
C03377=1152.321,119.309,-55.214,-178.966,6.646,148.917
C03378=1152.316,119.558,-55.233,-178.963,6.648,148.916
C03379=1152.311,119.807,-55.253,-178.960,6.650,148.916
C03380=1152.307,120.057,-55.272,-178.958,6.651,148.915
C03381=1152.301,120.305,-55.291,-178.955,6.653,148.915
C03382=1152.297,120.555,-55.311,-178.952,6.655,148.914
C03383=1152.292,120.805,-55.330,-178.949,6.656,148.914
C03384=1152.287,121.053,-55.350,-178.946,6.658,148.914
C03385=1152.283,121.303,-55.369,-178.943,6.660,148.913
C03386=1152.277,121.552,-55.388,-178.941,6.661,148.913
C03387=1152.273,121.801,-55.408,-178.938,6.663,148.912
C03388=1152.268,122.050,-55.428,-178.935,6.665,148.912
C03389=1152.264,122.299,-55.447,-178.933,6.666,148.912
C03390=1152.259,122.548,-55.466,-178.930,6.667,148.911
C03391=1152.253,122.797,-55.486,-178.928,6.669,148.911
C03392=1152.249,123.047,-55.505,-178.925,6.670,148.910
C03393=1152.244,123.296,-55.525,-178.922,6.672,148.910
C03394=1152.239,123.545,-55.544,-178.919,6.674,148.909
C03395=1152.234,123.795,-55.564,-178.916,6.676,148.909
C03396=1152.230,124.043,-55.584,-178.914,6.677,148.909
C03397=1152.225,124.292,-55.603,-178.911,6.679,148.908
C03398=1152.220,124.542,-55.623,-178.908,6.681,148.908
C03399=1152.215,124.791,-55.642,-178.906,6.682,148.907
C03400=1152.210,125.040,-55.662,-178.903,6.684,148.907
C03401=1152.206,125.289,-55.682,-178.900,6.686,148.907
C03402=1152.201,125.539,-55.702,-178.897,6.687,148.906
C03403=1152.196,125.788,-55.721,-178.894,6.689,148.906
C03404=1152.191,126.037,-55.741,-178.891,6.691,148.905
C03405=1152.187,126.286,-55.760,-178.889,6.692,148.905
C03406=1152.182,126.535,-55.780,-178.886,6.694,148.904
C03407=1152.177,126.784,-55.799,-178.883,6.696,148.904
C03408=1152.172,127.034,-55.819,-178.881,6.697,148.904
C03409=1152.168,127.283,-55.839,-178.878,6.699,148.903
C03410=1152.163,127.532,-55.859,-178.875,6.701,148.903
C03411=1152.158,127.781,-55.878,-178.872,6.702,148.902
C03412=1152.153,128.030,-55.899,-178.870,6.704,148.902
C03413=1152.148,128.280,-55.918,-178.867,6.706,148.902
C03414=1152.143,128.528,-55.938,-178.864,6.708,148.901
C03415=1152.139,128.777,-55.958,-178.862,6.709,148.901
C03416=1152.134,129.027,-55.978,-178.859,6.711,148.900
C03417=1152.130,129.276,-55.998,-178.856,6.713,148.900
C03418=1152.125,129.526,-56.018,-178.853,6.714,148.899
C03419=1152.119,129.774,-56.037,-178.850,6.716,148.899
C03420=1152.115,130.023,-56.057,-178.848,6.718,148.899
C03421=1152.110,130.273,-56.077,-178.845,6.719,148.898
C03422=1152.106,130.522,-56.097,-178.842,6.721,148.898
C03423=1152.100,130.771,-56.117,-178.839,6.723,148.897
C03424=1152.095,131.020,-56.138,-178.837,6.724,148.897
C03425=1152.091,131.270,-56.157,-178.834,6.726,148.897
C03426=1152.086,131.538,-56.178,-178.831,6.728,148.896
C03427=1152.080,131.807,-56.201,-178.828,6.730,148.896
C03428=1152.075,132.075,-56.222,-178.825,6.732,148.895
C03429=1152.070,132.344,-56.243,-178.822,6.733,148.895
C03430=1152.065,132.593,-56.264,-178.819,6.735,148.894
C03431=1152.061,132.843,-56.284,-178.817,6.737,148.894
C03432=1152.056,133.091,-56.304,-178.814,6.739,148.894
C03433=1152.051,133.340,-56.324,-178.811,6.740,148.893
C03434=1152.046,133.589,-56.344,-178.808,6.742,148.893
C03435=1152.042,133.838,-56.364,-178.806,6.744,148.892
C03436=1152.037,134.088,-56.384,-178.803,6.745,148.892
C03437=1152.032,134.337,-56.405,-178.800,6.748,148.892
C03438=1152.027,134.585,-56.425,-178.797,6.750,148.891
C03439=1152.022,134.835,-56.444,-178.794,6.751,148.891
C03440=1152.018,135.084,-56.465,-178.792,6.753,148.891
C03441=1152.013,135.333,-56.485,-178.789,6.755,148.890
C03442=1152.008,135.583,-56.505,-178.786,6.756,148.890
C03443=1152.003,135.832,-56.526,-178.783,6.758,148.889
C03444=1151.999,136.081,-56.546,-178.781,6.760,148.889
C03445=1151.994,136.330,-56.566,-178.778,6.762,148.889
C03446=1151.989,136.580,-56.587,-178.775,6.763,148.888
C03447=1151.984,136.828,-56.607,-178.773,6.765,148.888
C03448=1151.980,137.077,-56.627,-178.770,6.767,148.887
C03449=1151.975,137.326,-56.647,-178.767,6.768,148.887
C03450=1151.970,137.576,-56.668,-178.764,6.770,148.887
C03451=1151.965,137.824,-56.688,-178.762,6.772,148.886
C03452=1151.961,138.073,-56.708,-178.759,6.774,148.886
C03453=1151.956,138.323,-56.728,-178.756,6.776,148.885
C03454=1151.951,138.572,-56.749,-178.753,6.778,148.885
C03455=1151.946,138.821,-56.769,-178.750,6.780,148.885
C03456=1151.942,139.070,-56.790,-178.748,6.781,148.884
C03457=1151.937,139.319,-56.811,-178.745,6.783,148.884
C03458=1151.932,139.568,-56.831,-178.742,6.785,148.884
C03459=1151.928,139.818,-56.851,-178.739,6.786,148.883
C03460=1151.922,140.067,-56.872,-178.737,6.788,148.883
C03461=1151.918,140.316,-56.892,-178.734,6.790,148.882
C03462=1151.914,140.565,-56.912,-178.731,6.792,148.882
C03463=1151.908,140.814,-56.933,-178.729,6.793,148.882
C03464=1151.904,141.063,-56.954,-178.725,6.796,148.881
C03465=1151.899,141.313,-56.975,-178.723,6.798,148.881
C03466=1151.894,141.562,-56.995,-178.720,6.799,148.880
C03467=1151.890,141.810,-57.015,-178.717,6.801,148.880
C03468=1151.885,142.060,-57.036,-178.715,6.803,148.880
C03469=1151.880,142.309,-57.057,-178.712,6.804,148.879
C03470=1151.875,142.558,-57.078,-178.709,6.806,148.879
C03471=1151.871,142.807,-57.098,-178.706,6.808,148.879
C03472=1151.866,143.056,-57.119,-178.704,6.810,148.878
C03473=1151.861,143.305,-57.139,-178.701,6.811,148.878
C03474=1151.857,143.554,-57.160,-178.698,6.814,148.877
C03475=1151.851,143.803,-57.181,-178.695,6.816,148.877
C03476=1151.847,144.052,-57.201,-178.692,6.817,148.877
C03477=1151.842,144.302,-57.222,-178.690,6.819,148.876
C03478=1151.837,144.550,-57.243,-178.687,6.821,148.876
C03479=1151.832,144.800,-57.263,-178.685,6.823,148.876
C03480=1151.828,145.049,-57.284,-178.682,6.825,148.875
C03481=1151.823,145.298,-57.305,-178.679,6.826,148.875
C03482=1151.819,145.546,-57.326,-178.676,6.829,148.875
C03483=1151.814,145.796,-57.347,-178.673,6.831,148.874
C03484=1151.809,146.045,-57.368,-178.670,6.832,148.874
C03485=1151.804,146.294,-57.389,-178.668,6.834,148.873
C03486=1151.800,146.543,-57.409,-178.665,6.836,148.873
C03487=1151.795,146.793,-57.430,-178.662,6.837,148.873
C03488=1151.790,147.041,-57.452,-178.660,6.839,148.872
C03489=1151.785,147.290,-57.472,-178.656,6.842,148.872
C03490=1151.780,147.539,-57.493,-178.654,6.843,148.871
C03491=1151.776,147.788,-57.513,-178.651,6.845,148.871
C03492=1151.771,148.038,-57.535,-178.648,6.847,148.871
C03493=1151.766,148.287,-57.556,-178.646,6.849,148.870
C03494=1151.762,148.536,-57.577,-178.643,6.851,148.870
C03495=1151.757,148.785,-57.598,-178.641,6.852,148.870
C03496=1151.753,149.034,-57.619,-178.637,6.855,148.869
C03497=1151.747,149.283,-57.640,-178.635,6.857,148.869
C03498=1151.742,149.532,-57.661,-178.632,6.858,148.869
C03499=1151.738,149.782,-57.681,-178.629,6.860,148.868
C03500=1151.734,150.030,-57.703,-178.626,6.862,148.868
C03501=1151.728,150.280,-57.724,-178.624,6.864,148.867
C03502=1151.724,150.529,-57.744,-178.620,6.866,148.867
C03503=1151.719,150.777,-57.766,-178.618,6.868,148.867
C03504=1151.714,151.026,-57.787,-178.615,6.869,148.866
C03505=1151.710,151.276,-57.809,-178.612,6.871,148.866
C03506=1151.705,151.525,-57.830,-178.610,6.873,148.866
C03507=1151.700,151.774,-57.850,-178.607,6.875,148.865
C03508=1151.695,152.023,-57.872,-178.604,6.878,148.865
C03509=1151.691,152.272,-57.893,-178.601,6.879,148.865
C03510=1151.686,152.521,-57.915,-178.599,6.881,148.864
C03511=1151.681,152.770,-57.936,-178.596,6.883,148.864
C03512=1151.676,153.019,-57.957,-178.593,6.884,148.864
C03513=1151.672,153.268,-57.978,-178.590,6.887,148.863
C03514=1151.668,153.517,-58.000,-178.587,6.889,148.863
C03515=1151.663,153.766,-58.021,-178.585,6.891,148.863
C03516=1151.658,154.015,-58.042,-178.582,6.893,148.862
C03517=1151.652,154.264,-58.063,-178.580,6.894,148.862
C03518=1151.649,154.513,-58.085,-178.576,6.897,148.861
C03519=1151.644,154.763,-58.106,-178.574,6.899,148.861
C03520=1151.639,155.011,-58.127,-178.571,6.900,148.861
C03521=1151.634,155.261,-58.148,-178.568,6.902,148.860
C03522=1151.629,155.510,-58.170,-178.566,6.904,148.860
C03523=1151.625,155.758,-58.191,-178.562,6.906,148.860
C03524=1151.620,156.007,-58.212,-178.560,6.908,148.859
C03525=1151.616,156.257,-58.234,-178.557,6.910,148.859
C03526=1151.611,156.506,-58.255,-178.555,6.912,148.859
C03527=1151.606,156.755,-58.277,-178.552,6.914,148.858
C03528=1151.601,157.003,-58.299,-178.549,6.916,148.858
C03529=1151.596,157.253,-58.320,-178.546,6.918,148.858
C03530=1151.592,157.522,-58.344,-178.543,6.920,148.857
C03531=1151.586,157.791,-58.367,-178.540,6.922,148.857
C03532=1151.582,158.060,-58.390,-178.537,6.924,148.856
C03533=1151.577,158.329,-58.414,-178.534,6.926,148.856
C03534=1151.571,158.578,-58.435,-178.531,6.928,148.856
C03535=1151.566,158.827,-58.456,-178.529,6.930,148.856
C03536=1151.562,159.076,-58.479,-178.526,6.933,148.855
C03537=1151.558,159.324,-58.500,-178.523,6.934,148.855
C03538=1151.553,159.574,-58.521,-178.520,6.936,148.854
C03539=1151.549,159.823,-58.543,-178.518,6.938,148.854
C03540=1151.544,160.072,-58.564,-178.515,6.940,148.854
C03541=1151.539,160.320,-58.586,-178.512,6.942,148.854
C03542=1151.535,160.570,-58.608,-178.509,6.944,148.853
C03543=1151.529,160.819,-58.629,-178.507,6.946,148.853
C03544=1151.525,161.068,-58.651,-178.504,6.948,148.852
C03545=1151.520,161.317,-58.673,-178.501,6.950,148.852
C03546=1151.515,161.566,-58.694,-178.498,6.952,148.852
C03547=1151.511,161.815,-58.716,-178.496,6.954,148.852
C03548=1151.506,162.064,-58.738,-178.493,6.957,148.851
C03549=1151.502,162.313,-58.760,-178.490,6.958,148.851
C03550=1151.496,162.562,-58.782,-178.487,6.960,148.850
C03551=1151.492,162.810,-58.804,-178.484,6.962,148.850
C03552=1151.487,163.060,-58.826,-178.481,6.964,148.850
C03553=1151.482,163.308,-58.848,-178.479,6.966,148.850
C03554=1151.478,163.558,-58.869,-178.476,6.968,148.849
C03555=1151.473,163.807,-58.891,-178.474,6.970,148.849
C03556=1151.469,164.056,-58.913,-178.470,6.972,148.848
C03557=1151.464,164.305,-58.935,-178.468,6.974,148.848
C03558=1151.460,164.554,-58.957,-178.465,6.976,148.848
C03559=1151.455,164.803,-58.978,-178.463,6.978,148.848
C03560=1151.451,165.052,-59.001,-178.459,6.981,148.847
C03561=1151.445,165.301,-59.023,-178.457,6.982,148.847
C03562=1151.441,165.550,-59.045,-178.454,6.984,148.846
C03563=1151.436,165.799,-59.067,-178.451,6.987,148.846
C03564=1151.432,166.048,-59.089,-178.448,6.989,148.846
C03565=1151.427,166.297,-59.111,-178.446,6.990,148.846
C03566=1151.423,166.546,-59.133,-178.443,6.992,148.845
C03567=1151.417,166.795,-59.155,-178.440,6.995,148.845
C03568=1151.413,167.044,-59.177,-178.438,6.997,148.845
C03569=1151.408,167.293,-59.199,-178.435,6.998,148.844
C03570=1151.404,167.542,-59.222,-178.432,7.001,148.844
C03571=1151.399,167.790,-59.243,-178.429,7.003,148.844
C03572=1151.394,168.040,-59.266,-178.427,7.005,148.843
C03573=1151.389,168.289,-59.288,-178.423,7.007,148.843
C03574=1151.385,168.538,-59.310,-178.421,7.009,148.843
C03575=1151.380,168.787,-59.331,-178.418,7.011,148.842
C03576=1151.375,169.036,-59.355,-178.415,7.013,148.842
C03577=1151.370,169.284,-59.376,-178.412,7.015,148.842
C03578=1151.366,169.534,-59.399,-178.410,7.017,148.842
C03579=1151.361,169.782,-59.421,-178.407,7.019,148.841
C03580=1151.357,170.031,-59.444,-178.404,7.022,148.841
C03581=1151.352,170.281,-59.466,-178.402,7.024,148.841
C03582=1151.347,170.529,-59.487,-178.399,7.025,148.840
C03583=1151.343,170.778,-59.511,-178.396,7.028,148.840
C03584=1151.338,171.027,-59.532,-178.393,7.030,148.840
C03585=1151.334,171.276,-59.554,-178.391,7.032,148.839
C03586=1151.329,171.525,-59.578,-178.387,7.034,148.839
C03587=1151.324,171.774,-59.599,-178.385,7.036,148.839
C03588=1151.320,172.023,-59.621,-178.382,7.038,148.838
C03589=1151.315,172.272,-59.644,-178.379,7.041,148.838
C03590=1151.310,172.521,-59.667,-178.376,7.042,148.838
C03591=1151.306,172.770,-59.690,-178.374,7.044,148.837
C03592=1151.301,173.019,-59.712,-178.370,7.047,148.837
C03593=1151.296,173.268,-59.734,-178.368,7.049,148.837
C03594=1151.292,173.517,-59.757,-178.366,7.050,148.837
C03595=1151.287,173.766,-59.779,-178.362,7.053,148.836
C03596=1151.282,174.015,-59.802,-178.360,7.055,148.836
C03597=1151.278,174.264,-59.824,-178.357,7.057,148.836
C03598=1151.273,174.512,-59.847,-178.354,7.059,148.835
C03599=1151.268,174.762,-59.869,-178.351,7.061,148.835
C03600=1151.264,175.010,-59.892,-178.349,7.064,148.835
C03601=1151.259,175.259,-59.914,-178.346,7.066,148.835
C03602=1151.255,175.508,-59.937,-178.343,7.068,148.834
C03603=1151.250,175.758,-59.960,-178.340,7.070,148.834
C03604=1151.245,176.006,-59.982,-178.338,7.072,148.834
C03605=1151.240,176.255,-60.005,-178.335,7.074,148.833
C03606=1151.236,176.504,-60.027,-178.332,7.076,148.833
C03607=1151.231,176.752,-60.050,-178.330,7.079,148.833
C03608=1151.227,177.002,-60.072,-178.327,7.080,148.832
C03609=1151.222,177.251,-60.096,-178.324,7.083,148.832
C03610=1151.218,177.500,-60.118,-178.321,7.085,148.832
C03611=1151.212,177.748,-60.141,-178.318,7.087,148.832
C03612=1151.208,177.997,-60.164,-178.315,7.089,148.831
C03613=1151.203,178.247,-60.186,-178.313,7.091,148.831
C03614=1151.199,178.496,-60.210,-178.310,7.094,148.831
C03615=1151.194,178.744,-60.232,-178.307,7.096,148.830
C03616=1151.189,178.993,-60.255,-178.304,7.097,148.830
C03617=1151.185,179.242,-60.277,-178.302,7.100,148.830
C03618=1151.180,179.491,-60.301,-178.299,7.102,148.830
C03619=1151.176,179.739,-60.323,-178.296,7.105,148.829
C03620=1151.171,179.989,-60.346,-178.293,7.107,148.829
C03621=1151.166,180.238,-60.369,-178.291,7.108,148.829
C03622=1151.162,180.487,-60.392,-178.288,7.111,148.828
C03623=1151.158,180.736,-60.415,-178.285,7.113,148.828
C03624=1151.152,180.984,-60.438,-178.282,7.116,148.828
C03625=1151.148,181.233,-60.460,-178.279,7.117,148.828
C03626=1151.143,181.482,-60.484,-178.277,7.119,148.827
C03627=1151.139,181.731,-60.507,-178.274,7.122,148.827
C03628=1151.135,181.980,-60.530,-178.271,7.124,148.827
C03629=1151.129,182.229,-60.553,-178.268,7.127,148.827
C03630=1151.125,182.478,-60.576,-178.266,7.128,148.826
C03631=1151.121,182.726,-60.599,-178.262,7.131,148.826
C03632=1151.116,182.976,-60.622,-178.260,7.133,148.826
C03633=1151.111,183.225,-60.645,-178.257,7.135,148.825
C03634=1151.107,183.494,-60.670,-178.254,7.137,148.825
C03635=1151.101,183.764,-60.695,-178.251,7.140,148.825
C03636=1151.096,184.033,-60.720,-178.249,7.142,148.825
C03637=1151.091,184.303,-60.745,-178.245,7.145,148.824
C03638=1151.087,184.552,-60.768,-178.242,7.147,148.824
C03639=1151.082,184.801,-60.791,-178.240,7.149,148.824
C03640=1151.077,185.050,-60.815,-178.237,7.151,148.823
C03641=1151.073,185.299,-60.838,-178.234,7.154,148.823
C03642=1151.069,185.548,-60.861,-178.232,7.156,148.823
C03643=1151.064,185.797,-60.884,-178.228,7.158,148.823
C03644=1151.059,186.045,-60.907,-178.226,7.160,148.822
C03645=1151.054,186.294,-60.930,-178.223,7.163,148.822
C03646=1151.049,186.543,-60.954,-178.220,7.165,148.822
C03647=1151.045,186.792,-60.977,-178.217,7.167,148.822
C03648=1151.041,187.040,-61.001,-178.215,7.169,148.821
C03649=1151.036,187.289,-61.024,-178.213,7.171,148.821
C03650=1151.032,187.538,-61.047,-178.209,7.174,148.821
C03651=1151.027,187.787,-61.071,-178.207,7.176,148.820
C03652=1151.022,188.036,-61.094,-178.204,7.179,148.820
C03653=1151.017,188.285,-61.117,-178.201,7.180,148.820
C03654=1151.013,188.534,-61.141,-178.198,7.183,148.820
C03655=1151.008,188.783,-61.165,-178.196,7.185,148.819
C03656=1151.004,189.032,-61.188,-178.192,7.187,148.819
C03657=1151.000,189.281,-61.211,-178.190,7.190,148.819
C03658=1150.995,189.530,-61.234,-178.187,7.192,148.819
C03659=1150.990,189.779,-61.258,-178.185,7.194,148.818
C03660=1150.986,190.027,-61.282,-178.181,7.197,148.818
C03661=1150.981,190.276,-61.305,-178.179,7.199,148.818
C03662=1150.976,190.524,-61.328,-178.176,7.201,148.818
